   // GBK_TO_UNICODE[12068] := 16#A0D0;
   // GBK_TO_UNICODE[12069] := 16#7298;
   // GBK_TO_UNICODE[12070] := 16#A0D1;
   // GBK_TO_UNICODE[12071] := 16#7299;
   // GBK_TO_UNICODE[12072] := 16#A0D2;
   // GBK_TO_UNICODE[12073] := 16#729A;
   // GBK_TO_UNICODE[12074] := 16#A0D3;
   // GBK_TO_UNICODE[12075] := 16#729B;
   // GBK_TO_UNICODE[12076] := 16#A0D4;
   // GBK_TO_UNICODE[12077] := 16#729C;
   // GBK_TO_UNICODE[12078] := 16#A0D5;
   // GBK_TO_UNICODE[12079] := 16#729D;
   // GBK_TO_UNICODE[12080] := 16#A0D6;
   // GBK_TO_UNICODE[12081] := 16#729E;
   // GBK_TO_UNICODE[12082] := 16#A0D7;
   // GBK_TO_UNICODE[12083] := 16#72A0;
   // GBK_TO_UNICODE[12084] := 16#A0D8;
   // GBK_TO_UNICODE[12085] := 16#72A1;
   // GBK_TO_UNICODE[12086] := 16#A0D9;
   // GBK_TO_UNICODE[12087] := 16#72A2;
   // GBK_TO_UNICODE[12088] := 16#A0DA;
   // GBK_TO_UNICODE[12089] := 16#72A3;
   // GBK_TO_UNICODE[12090] := 16#A0DB;
   // GBK_TO_UNICODE[12091] := 16#72A4;
   // GBK_TO_UNICODE[12092] := 16#A0DC;
   // GBK_TO_UNICODE[12093] := 16#72A5;
   // GBK_TO_UNICODE[12094] := 16#A0DD;
   // GBK_TO_UNICODE[12095] := 16#72A6;
   // GBK_TO_UNICODE[12096] := 16#A0DE;
   // GBK_TO_UNICODE[12097] := 16#72A7;
   // GBK_TO_UNICODE[12098] := 16#A0DF;
   // GBK_TO_UNICODE[12099] := 16#72A8;
   // GBK_TO_UNICODE[12100] := 16#A0E0;
   // GBK_TO_UNICODE[12101] := 16#72A9;
   // GBK_TO_UNICODE[12102] := 16#A0E1;
   // GBK_TO_UNICODE[12103] := 16#72AA;
   // GBK_TO_UNICODE[12104] := 16#A0E2;
   // GBK_TO_UNICODE[12105] := 16#72AB;
   // GBK_TO_UNICODE[12106] := 16#A0E3;
   // GBK_TO_UNICODE[12107] := 16#72AE;
   // GBK_TO_UNICODE[12108] := 16#A0E4;
   // GBK_TO_UNICODE[12109] := 16#72B1;
   // GBK_TO_UNICODE[12110] := 16#A0E5;
   // GBK_TO_UNICODE[12111] := 16#72B2;
   // GBK_TO_UNICODE[12112] := 16#A0E6;
   // GBK_TO_UNICODE[12113] := 16#72B3;
   // GBK_TO_UNICODE[12114] := 16#A0E7;
   // GBK_TO_UNICODE[12115] := 16#72B5;
   // GBK_TO_UNICODE[12116] := 16#A0E8;
   // GBK_TO_UNICODE[12117] := 16#72BA;
   // GBK_TO_UNICODE[12118] := 16#A0E9;
   // GBK_TO_UNICODE[12119] := 16#72BB;
   // GBK_TO_UNICODE[12120] := 16#A0EA;
   // GBK_TO_UNICODE[12121] := 16#72BC;
   // GBK_TO_UNICODE[12122] := 16#A0EB;
   // GBK_TO_UNICODE[12123] := 16#72BD;
   // GBK_TO_UNICODE[12124] := 16#A0EC;
   // GBK_TO_UNICODE[12125] := 16#72BE;
   // GBK_TO_UNICODE[12126] := 16#A0ED;
   // GBK_TO_UNICODE[12127] := 16#72BF;
   // GBK_TO_UNICODE[12128] := 16#A0EE;
   // GBK_TO_UNICODE[12129] := 16#72C0;
   // GBK_TO_UNICODE[12130] := 16#A0EF;
   // GBK_TO_UNICODE[12131] := 16#72C5;
   // GBK_TO_UNICODE[12132] := 16#A0F0;
   // GBK_TO_UNICODE[12133] := 16#72C6;
   // GBK_TO_UNICODE[12134] := 16#A0F1;
   // GBK_TO_UNICODE[12135] := 16#72C7;
   // GBK_TO_UNICODE[12136] := 16#A0F2;
   // GBK_TO_UNICODE[12137] := 16#72C9;
   // GBK_TO_UNICODE[12138] := 16#A0F3;
   // GBK_TO_UNICODE[12139] := 16#72CA;
   // GBK_TO_UNICODE[12140] := 16#A0F4;
   // GBK_TO_UNICODE[12141] := 16#72CB;
   // GBK_TO_UNICODE[12142] := 16#A0F5;
   // GBK_TO_UNICODE[12143] := 16#72CC;
   // GBK_TO_UNICODE[12144] := 16#A0F6;
   // GBK_TO_UNICODE[12145] := 16#72CF;
   // GBK_TO_UNICODE[12146] := 16#A0F7;
   // GBK_TO_UNICODE[12147] := 16#72D1;
   // GBK_TO_UNICODE[12148] := 16#A0F8;
   // GBK_TO_UNICODE[12149] := 16#72D3;
   // GBK_TO_UNICODE[12150] := 16#A0F9;
   // GBK_TO_UNICODE[12151] := 16#72D4;
   // GBK_TO_UNICODE[12152] := 16#A0FA;
   // GBK_TO_UNICODE[12153] := 16#72D5;
   // GBK_TO_UNICODE[12154] := 16#A0FB;
   // GBK_TO_UNICODE[12155] := 16#72D6;
   // GBK_TO_UNICODE[12156] := 16#A0FC;
   // GBK_TO_UNICODE[12157] := 16#72D8;
   // GBK_TO_UNICODE[12158] := 16#A0FD;
   // GBK_TO_UNICODE[12159] := 16#72DA;
   // GBK_TO_UNICODE[12160] := 16#A0FE;
   // GBK_TO_UNICODE[12161] := 16#72DB;
   // GBK_TO_UNICODE[12162] := 16#A1A1;
   // GBK_TO_UNICODE[12163] := 16#3000;
   // GBK_TO_UNICODE[12164] := 16#A1A2;
   // GBK_TO_UNICODE[12165] := 16#3001;
   // GBK_TO_UNICODE[12166] := 16#A1A3;
   // GBK_TO_UNICODE[12167] := 16#3002;
   // GBK_TO_UNICODE[12168] := 16#A1A4;
   // GBK_TO_UNICODE[12169] := 16#00B7;
   // GBK_TO_UNICODE[12170] := 16#A1A5;
   // GBK_TO_UNICODE[12171] := 16#02C9;
   // GBK_TO_UNICODE[12172] := 16#A1A6;
   // GBK_TO_UNICODE[12173] := 16#02C7;
   // GBK_TO_UNICODE[12174] := 16#A1A7;
   // GBK_TO_UNICODE[12175] := 16#00A8;
   // GBK_TO_UNICODE[12176] := 16#A1A8;
   // GBK_TO_UNICODE[12177] := 16#3003;
   // GBK_TO_UNICODE[12178] := 16#A1A9;
   // GBK_TO_UNICODE[12179] := 16#3005;
   // GBK_TO_UNICODE[12180] := 16#A1AA;
   // GBK_TO_UNICODE[12181] := 16#2014;
   // GBK_TO_UNICODE[12182] := 16#A1AB;
   // GBK_TO_UNICODE[12183] := 16#FF5E;
   // GBK_TO_UNICODE[12184] := 16#A1AC;
   // GBK_TO_UNICODE[12185] := 16#2016;
   // GBK_TO_UNICODE[12186] := 16#A1AD;
   // GBK_TO_UNICODE[12187] := 16#2026;
   // GBK_TO_UNICODE[12188] := 16#A1AE;
   // GBK_TO_UNICODE[12189] := 16#2018;
   // GBK_TO_UNICODE[12190] := 16#A1AF;
   // GBK_TO_UNICODE[12191] := 16#2019;
   // GBK_TO_UNICODE[12192] := 16#A1B0;
   // GBK_TO_UNICODE[12193] := 16#201C;
   // GBK_TO_UNICODE[12194] := 16#A1B1;
   // GBK_TO_UNICODE[12195] := 16#201D;
   // GBK_TO_UNICODE[12196] := 16#A1B2;
   // GBK_TO_UNICODE[12197] := 16#3014;
   // GBK_TO_UNICODE[12198] := 16#A1B3;
   // GBK_TO_UNICODE[12199] := 16#3015;
   // GBK_TO_UNICODE[12200] := 16#A1B4;
   // GBK_TO_UNICODE[12201] := 16#3008;
   // GBK_TO_UNICODE[12202] := 16#A1B5;
   // GBK_TO_UNICODE[12203] := 16#3009;
   // GBK_TO_UNICODE[12204] := 16#A1B6;
   // GBK_TO_UNICODE[12205] := 16#300A;
   // GBK_TO_UNICODE[12206] := 16#A1B7;
   // GBK_TO_UNICODE[12207] := 16#300B;
   // GBK_TO_UNICODE[12208] := 16#A1B8;
   // GBK_TO_UNICODE[12209] := 16#300C;
   // GBK_TO_UNICODE[12210] := 16#A1B9;
   // GBK_TO_UNICODE[12211] := 16#300D;
   // GBK_TO_UNICODE[12212] := 16#A1BA;
   // GBK_TO_UNICODE[12213] := 16#300E;
   // GBK_TO_UNICODE[12214] := 16#A1BB;
   // GBK_TO_UNICODE[12215] := 16#300F;
   // GBK_TO_UNICODE[12216] := 16#A1BC;
   // GBK_TO_UNICODE[12217] := 16#3016;
   // GBK_TO_UNICODE[12218] := 16#A1BD;
   // GBK_TO_UNICODE[12219] := 16#3017;
   // GBK_TO_UNICODE[12220] := 16#A1BE;
   // GBK_TO_UNICODE[12221] := 16#3010;
   // GBK_TO_UNICODE[12222] := 16#A1BF;
   // GBK_TO_UNICODE[12223] := 16#3011;
   // GBK_TO_UNICODE[12224] := 16#A1C0;
   // GBK_TO_UNICODE[12225] := 16#00B1;
   // GBK_TO_UNICODE[12226] := 16#A1C1;
   // GBK_TO_UNICODE[12227] := 16#00D7;
   // GBK_TO_UNICODE[12228] := 16#A1C2;
   // GBK_TO_UNICODE[12229] := 16#00F7;
   // GBK_TO_UNICODE[12230] := 16#A1C3;
   // GBK_TO_UNICODE[12231] := 16#2236;
   // GBK_TO_UNICODE[12232] := 16#A1C4;
   // GBK_TO_UNICODE[12233] := 16#2227;
   // GBK_TO_UNICODE[12234] := 16#A1C5;
   // GBK_TO_UNICODE[12235] := 16#2228;
   // GBK_TO_UNICODE[12236] := 16#A1C6;
   // GBK_TO_UNICODE[12237] := 16#2211;
   // GBK_TO_UNICODE[12238] := 16#A1C7;
   // GBK_TO_UNICODE[12239] := 16#220F;
   // GBK_TO_UNICODE[12240] := 16#A1C8;
   // GBK_TO_UNICODE[12241] := 16#222A;
   // GBK_TO_UNICODE[12242] := 16#A1C9;
   // GBK_TO_UNICODE[12243] := 16#2229;
   // GBK_TO_UNICODE[12244] := 16#A1CA;
   // GBK_TO_UNICODE[12245] := 16#2208;
   // GBK_TO_UNICODE[12246] := 16#A1CB;
   // GBK_TO_UNICODE[12247] := 16#2237;
   // GBK_TO_UNICODE[12248] := 16#A1CC;
   // GBK_TO_UNICODE[12249] := 16#221A;
   // GBK_TO_UNICODE[12250] := 16#A1CD;
   // GBK_TO_UNICODE[12251] := 16#22A5;
   // GBK_TO_UNICODE[12252] := 16#A1CE;
   // GBK_TO_UNICODE[12253] := 16#2225;
   // GBK_TO_UNICODE[12254] := 16#A1CF;
   // GBK_TO_UNICODE[12255] := 16#2220;
   // GBK_TO_UNICODE[12256] := 16#A1D0;
   // GBK_TO_UNICODE[12257] := 16#2312;
   // GBK_TO_UNICODE[12258] := 16#A1D1;
   // GBK_TO_UNICODE[12259] := 16#2299;
   // GBK_TO_UNICODE[12260] := 16#A1D2;
   // GBK_TO_UNICODE[12261] := 16#222B;
   // GBK_TO_UNICODE[12262] := 16#A1D3;
   // GBK_TO_UNICODE[12263] := 16#222E;
   // GBK_TO_UNICODE[12264] := 16#A1D4;
   // GBK_TO_UNICODE[12265] := 16#2261;
   // GBK_TO_UNICODE[12266] := 16#A1D5;
   // GBK_TO_UNICODE[12267] := 16#224C;
   // GBK_TO_UNICODE[12268] := 16#A1D6;
   // GBK_TO_UNICODE[12269] := 16#2248;
   // GBK_TO_UNICODE[12270] := 16#A1D7;
   // GBK_TO_UNICODE[12271] := 16#223D;
   // GBK_TO_UNICODE[12272] := 16#A1D8;
   // GBK_TO_UNICODE[12273] := 16#221D;
   // GBK_TO_UNICODE[12274] := 16#A1D9;
   // GBK_TO_UNICODE[12275] := 16#2260;
   // GBK_TO_UNICODE[12276] := 16#A1DA;
   // GBK_TO_UNICODE[12277] := 16#226E;
   // GBK_TO_UNICODE[12278] := 16#A1DB;
   // GBK_TO_UNICODE[12279] := 16#226F;
   // GBK_TO_UNICODE[12280] := 16#A1DC;
   // GBK_TO_UNICODE[12281] := 16#2264;
   // GBK_TO_UNICODE[12282] := 16#A1DD;
   // GBK_TO_UNICODE[12283] := 16#2265;
   // GBK_TO_UNICODE[12284] := 16#A1DE;
   // GBK_TO_UNICODE[12285] := 16#221E;
   // GBK_TO_UNICODE[12286] := 16#A1DF;
   // GBK_TO_UNICODE[12287] := 16#2235;
   // GBK_TO_UNICODE[12288] := 16#A1E0;
   // GBK_TO_UNICODE[12289] := 16#2234;
   // GBK_TO_UNICODE[12290] := 16#A1E1;
   // GBK_TO_UNICODE[12291] := 16#2642;
   // GBK_TO_UNICODE[12292] := 16#A1E2;
   // GBK_TO_UNICODE[12293] := 16#2640;
   // GBK_TO_UNICODE[12294] := 16#A1E3;
   // GBK_TO_UNICODE[12295] := 16#00B0;
   // GBK_TO_UNICODE[12296] := 16#A1E4;
   // GBK_TO_UNICODE[12297] := 16#2032;
   // GBK_TO_UNICODE[12298] := 16#A1E5;
   // GBK_TO_UNICODE[12299] := 16#2033;
   // GBK_TO_UNICODE[12300] := 16#A1E6;
   // GBK_TO_UNICODE[12301] := 16#2103;
   // GBK_TO_UNICODE[12302] := 16#A1E7;
   // GBK_TO_UNICODE[12303] := 16#FF04;
   // GBK_TO_UNICODE[12304] := 16#A1E8;
   // GBK_TO_UNICODE[12305] := 16#00A4;
   // GBK_TO_UNICODE[12306] := 16#A1E9;
   // GBK_TO_UNICODE[12307] := 16#FFE0;
   // GBK_TO_UNICODE[12308] := 16#A1EA;
   // GBK_TO_UNICODE[12309] := 16#FFE1;
   // GBK_TO_UNICODE[12310] := 16#A1EB;
   // GBK_TO_UNICODE[12311] := 16#2030;
   // GBK_TO_UNICODE[12312] := 16#A1EC;
   // GBK_TO_UNICODE[12313] := 16#00A7;
   // GBK_TO_UNICODE[12314] := 16#A1ED;
   // GBK_TO_UNICODE[12315] := 16#2116;
   // GBK_TO_UNICODE[12316] := 16#A1EE;
   // GBK_TO_UNICODE[12317] := 16#2606;
   // GBK_TO_UNICODE[12318] := 16#A1EF;
   // GBK_TO_UNICODE[12319] := 16#2605;
   // GBK_TO_UNICODE[12320] := 16#A1F0;
   // GBK_TO_UNICODE[12321] := 16#25CB;
   // GBK_TO_UNICODE[12322] := 16#A1F1;
   // GBK_TO_UNICODE[12323] := 16#25CF;
   // GBK_TO_UNICODE[12324] := 16#A1F2;
   // GBK_TO_UNICODE[12325] := 16#25CE;
   // GBK_TO_UNICODE[12326] := 16#A1F3;
   // GBK_TO_UNICODE[12327] := 16#25C7;
   // GBK_TO_UNICODE[12328] := 16#A1F4;
   // GBK_TO_UNICODE[12329] := 16#25C6;
   // GBK_TO_UNICODE[12330] := 16#A1F5;
   // GBK_TO_UNICODE[12331] := 16#25A1;
   // GBK_TO_UNICODE[12332] := 16#A1F6;
   // GBK_TO_UNICODE[12333] := 16#25A0;
   // GBK_TO_UNICODE[12334] := 16#A1F7;
   // GBK_TO_UNICODE[12335] := 16#25B3;
   // GBK_TO_UNICODE[12336] := 16#A1F8;
   // GBK_TO_UNICODE[12337] := 16#25B2;
   // GBK_TO_UNICODE[12338] := 16#A1F9;
   // GBK_TO_UNICODE[12339] := 16#203B;
   // GBK_TO_UNICODE[12340] := 16#A1FA;
   // GBK_TO_UNICODE[12341] := 16#2192;
   // GBK_TO_UNICODE[12342] := 16#A1FB;
   // GBK_TO_UNICODE[12343] := 16#2190;
   // GBK_TO_UNICODE[12344] := 16#A1FC;
   // GBK_TO_UNICODE[12345] := 16#2191;
   // GBK_TO_UNICODE[12346] := 16#A1FD;
   // GBK_TO_UNICODE[12347] := 16#2193;
   // GBK_TO_UNICODE[12348] := 16#A1FE;
   // GBK_TO_UNICODE[12349] := 16#3013;
   // GBK_TO_UNICODE[12350] := 16#A2A1;
   // GBK_TO_UNICODE[12351] := 16#2170;
   // GBK_TO_UNICODE[12352] := 16#A2A2;
   // GBK_TO_UNICODE[12353] := 16#2171;
   // GBK_TO_UNICODE[12354] := 16#A2A3;
   // GBK_TO_UNICODE[12355] := 16#2172;
   // GBK_TO_UNICODE[12356] := 16#A2A4;
   // GBK_TO_UNICODE[12357] := 16#2173;
   // GBK_TO_UNICODE[12358] := 16#A2A5;
   // GBK_TO_UNICODE[12359] := 16#2174;
   // GBK_TO_UNICODE[12360] := 16#A2A6;
   // GBK_TO_UNICODE[12361] := 16#2175;
   // GBK_TO_UNICODE[12362] := 16#A2A7;
   // GBK_TO_UNICODE[12363] := 16#2176;
   // GBK_TO_UNICODE[12364] := 16#A2A8;
   // GBK_TO_UNICODE[12365] := 16#2177;
   // GBK_TO_UNICODE[12366] := 16#A2A9;
   // GBK_TO_UNICODE[12367] := 16#2178;
   // GBK_TO_UNICODE[12368] := 16#A2AA;
   // GBK_TO_UNICODE[12369] := 16#2179;
   // GBK_TO_UNICODE[12370] := 16#A2B1;
   // GBK_TO_UNICODE[12371] := 16#2488;
   // GBK_TO_UNICODE[12372] := 16#A2B2;
   // GBK_TO_UNICODE[12373] := 16#2489;
   // GBK_TO_UNICODE[12374] := 16#A2B3;
   // GBK_TO_UNICODE[12375] := 16#248A;
   // GBK_TO_UNICODE[12376] := 16#A2B4;
   // GBK_TO_UNICODE[12377] := 16#248B;
   // GBK_TO_UNICODE[12378] := 16#A2B5;
   // GBK_TO_UNICODE[12379] := 16#248C;
   // GBK_TO_UNICODE[12380] := 16#A2B6;
   // GBK_TO_UNICODE[12381] := 16#248D;
   // GBK_TO_UNICODE[12382] := 16#A2B7;
   // GBK_TO_UNICODE[12383] := 16#248E;
   // GBK_TO_UNICODE[12384] := 16#A2B8;
   // GBK_TO_UNICODE[12385] := 16#248F;
   // GBK_TO_UNICODE[12386] := 16#A2B9;
   // GBK_TO_UNICODE[12387] := 16#2490;
   // GBK_TO_UNICODE[12388] := 16#A2BA;
   // GBK_TO_UNICODE[12389] := 16#2491;
   // GBK_TO_UNICODE[12390] := 16#A2BB;
   // GBK_TO_UNICODE[12391] := 16#2492;
   // GBK_TO_UNICODE[12392] := 16#A2BC;
   // GBK_TO_UNICODE[12393] := 16#2493;
   // GBK_TO_UNICODE[12394] := 16#A2BD;
   // GBK_TO_UNICODE[12395] := 16#2494;
   // GBK_TO_UNICODE[12396] := 16#A2BE;
   // GBK_TO_UNICODE[12397] := 16#2495;
   // GBK_TO_UNICODE[12398] := 16#A2BF;
   // GBK_TO_UNICODE[12399] := 16#2496;
   // GBK_TO_UNICODE[12400] := 16#A2C0;
   // GBK_TO_UNICODE[12401] := 16#2497;
   // GBK_TO_UNICODE[12402] := 16#A2C1;
   // GBK_TO_UNICODE[12403] := 16#2498;
   // GBK_TO_UNICODE[12404] := 16#A2C2;
   // GBK_TO_UNICODE[12405] := 16#2499;
   // GBK_TO_UNICODE[12406] := 16#A2C3;
   // GBK_TO_UNICODE[12407] := 16#249A;
   // GBK_TO_UNICODE[12408] := 16#A2C4;
   // GBK_TO_UNICODE[12409] := 16#249B;
   // GBK_TO_UNICODE[12410] := 16#A2C5;
   // GBK_TO_UNICODE[12411] := 16#2474;
   // GBK_TO_UNICODE[12412] := 16#A2C6;
   // GBK_TO_UNICODE[12413] := 16#2475;
   // GBK_TO_UNICODE[12414] := 16#A2C7;
   // GBK_TO_UNICODE[12415] := 16#2476;
   // GBK_TO_UNICODE[12416] := 16#A2C8;
   // GBK_TO_UNICODE[12417] := 16#2477;
   // GBK_TO_UNICODE[12418] := 16#A2C9;
   // GBK_TO_UNICODE[12419] := 16#2478;
   // GBK_TO_UNICODE[12420] := 16#A2CA;
   // GBK_TO_UNICODE[12421] := 16#2479;
   // GBK_TO_UNICODE[12422] := 16#A2CB;
   // GBK_TO_UNICODE[12423] := 16#247A;
   // GBK_TO_UNICODE[12424] := 16#A2CC;
   // GBK_TO_UNICODE[12425] := 16#247B;
   // GBK_TO_UNICODE[12426] := 16#A2CD;
   // GBK_TO_UNICODE[12427] := 16#247C;
   // GBK_TO_UNICODE[12428] := 16#A2CE;
   // GBK_TO_UNICODE[12429] := 16#247D;
   // GBK_TO_UNICODE[12430] := 16#A2CF;
   // GBK_TO_UNICODE[12431] := 16#247E;
   // GBK_TO_UNICODE[12432] := 16#A2D0;
   // GBK_TO_UNICODE[12433] := 16#247F;
   // GBK_TO_UNICODE[12434] := 16#A2D1;
   // GBK_TO_UNICODE[12435] := 16#2480;
   // GBK_TO_UNICODE[12436] := 16#A2D2;
   // GBK_TO_UNICODE[12437] := 16#2481;
   // GBK_TO_UNICODE[12438] := 16#A2D3;
   // GBK_TO_UNICODE[12439] := 16#2482;
   // GBK_TO_UNICODE[12440] := 16#A2D4;
   // GBK_TO_UNICODE[12441] := 16#2483;
   // GBK_TO_UNICODE[12442] := 16#A2D5;
   // GBK_TO_UNICODE[12443] := 16#2484;
   // GBK_TO_UNICODE[12444] := 16#A2D6;
   // GBK_TO_UNICODE[12445] := 16#2485;
   // GBK_TO_UNICODE[12446] := 16#A2D7;
   // GBK_TO_UNICODE[12447] := 16#2486;
   // GBK_TO_UNICODE[12448] := 16#A2D8;
   // GBK_TO_UNICODE[12449] := 16#2487;
   // GBK_TO_UNICODE[12450] := 16#A2D9;
   // GBK_TO_UNICODE[12451] := 16#2460;
   // GBK_TO_UNICODE[12452] := 16#A2DA;
   // GBK_TO_UNICODE[12453] := 16#2461;
   // GBK_TO_UNICODE[12454] := 16#A2DB;
   // GBK_TO_UNICODE[12455] := 16#2462;
   // GBK_TO_UNICODE[12456] := 16#A2DC;
   // GBK_TO_UNICODE[12457] := 16#2463;
   // GBK_TO_UNICODE[12458] := 16#A2DD;
   // GBK_TO_UNICODE[12459] := 16#2464;
   // GBK_TO_UNICODE[12460] := 16#A2DE;
   // GBK_TO_UNICODE[12461] := 16#2465;
   // GBK_TO_UNICODE[12462] := 16#A2DF;
   // GBK_TO_UNICODE[12463] := 16#2466;
   // GBK_TO_UNICODE[12464] := 16#A2E0;
   // GBK_TO_UNICODE[12465] := 16#2467;
   // GBK_TO_UNICODE[12466] := 16#A2E1;
   // GBK_TO_UNICODE[12467] := 16#2468;
   // GBK_TO_UNICODE[12468] := 16#A2E2;
   // GBK_TO_UNICODE[12469] := 16#2469;
   // GBK_TO_UNICODE[12470] := 16#A2E5;
   // GBK_TO_UNICODE[12471] := 16#3220;
   // GBK_TO_UNICODE[12472] := 16#A2E6;
   // GBK_TO_UNICODE[12473] := 16#3221;
   // GBK_TO_UNICODE[12474] := 16#A2E7;
   // GBK_TO_UNICODE[12475] := 16#3222;
   // GBK_TO_UNICODE[12476] := 16#A2E8;
   // GBK_TO_UNICODE[12477] := 16#3223;
   // GBK_TO_UNICODE[12478] := 16#A2E9;
   // GBK_TO_UNICODE[12479] := 16#3224;
   // GBK_TO_UNICODE[12480] := 16#A2EA;
   // GBK_TO_UNICODE[12481] := 16#3225;
   // GBK_TO_UNICODE[12482] := 16#A2EB;
   // GBK_TO_UNICODE[12483] := 16#3226;
   // GBK_TO_UNICODE[12484] := 16#A2EC;
   // GBK_TO_UNICODE[12485] := 16#3227;
   // GBK_TO_UNICODE[12486] := 16#A2ED;
   // GBK_TO_UNICODE[12487] := 16#3228;
   // GBK_TO_UNICODE[12488] := 16#A2EE;
   // GBK_TO_UNICODE[12489] := 16#3229;
   // GBK_TO_UNICODE[12490] := 16#A2F1;
   // GBK_TO_UNICODE[12491] := 16#2160;
   // GBK_TO_UNICODE[12492] := 16#A2F2;
   // GBK_TO_UNICODE[12493] := 16#2161;
   // GBK_TO_UNICODE[12494] := 16#A2F3;
   // GBK_TO_UNICODE[12495] := 16#2162;
   // GBK_TO_UNICODE[12496] := 16#A2F4;
   // GBK_TO_UNICODE[12497] := 16#2163;
   // GBK_TO_UNICODE[12498] := 16#A2F5;
   // GBK_TO_UNICODE[12499] := 16#2164;
   // GBK_TO_UNICODE[12500] := 16#A2F6;
   // GBK_TO_UNICODE[12501] := 16#2165;
   // GBK_TO_UNICODE[12502] := 16#A2F7;
   // GBK_TO_UNICODE[12503] := 16#2166;
   // GBK_TO_UNICODE[12504] := 16#A2F8;
   // GBK_TO_UNICODE[12505] := 16#2167;
   // GBK_TO_UNICODE[12506] := 16#A2F9;
   // GBK_TO_UNICODE[12507] := 16#2168;
   // GBK_TO_UNICODE[12508] := 16#A2FA;
   // GBK_TO_UNICODE[12509] := 16#2169;
   // GBK_TO_UNICODE[12510] := 16#A2FB;
   // GBK_TO_UNICODE[12511] := 16#216A;
   // GBK_TO_UNICODE[12512] := 16#A2FC;
   // GBK_TO_UNICODE[12513] := 16#216B;
   // GBK_TO_UNICODE[12514] := 16#A3A1;
   // GBK_TO_UNICODE[12515] := 16#FF01;
   // GBK_TO_UNICODE[12516] := 16#A3A2;
   // GBK_TO_UNICODE[12517] := 16#FF02;
   // GBK_TO_UNICODE[12518] := 16#A3A3;
   // GBK_TO_UNICODE[12519] := 16#FF03;
   // GBK_TO_UNICODE[12520] := 16#A3A4;
   // GBK_TO_UNICODE[12521] := 16#FFE5;
   // GBK_TO_UNICODE[12522] := 16#A3A5;
   // GBK_TO_UNICODE[12523] := 16#FF05;
   // GBK_TO_UNICODE[12524] := 16#A3A6;
   // GBK_TO_UNICODE[12525] := 16#FF06;
   // GBK_TO_UNICODE[12526] := 16#A3A7;
   // GBK_TO_UNICODE[12527] := 16#FF07;
   // GBK_TO_UNICODE[12528] := 16#A3A8;
   // GBK_TO_UNICODE[12529] := 16#FF08;
   // GBK_TO_UNICODE[12530] := 16#A3A9;
   // GBK_TO_UNICODE[12531] := 16#FF09;
   // GBK_TO_UNICODE[12532] := 16#A3AA;
   // GBK_TO_UNICODE[12533] := 16#FF0A;
   // GBK_TO_UNICODE[12534] := 16#A3AB;
   // GBK_TO_UNICODE[12535] := 16#FF0B;
   // GBK_TO_UNICODE[12536] := 16#A3AC;
   // GBK_TO_UNICODE[12537] := 16#FF0C;
   // GBK_TO_UNICODE[12538] := 16#A3AD;
   // GBK_TO_UNICODE[12539] := 16#FF0D;
   // GBK_TO_UNICODE[12540] := 16#A3AE;
   // GBK_TO_UNICODE[12541] := 16#FF0E;
   // GBK_TO_UNICODE[12542] := 16#A3AF;
   // GBK_TO_UNICODE[12543] := 16#FF0F;
   // GBK_TO_UNICODE[12544] := 16#A3B0;
   // GBK_TO_UNICODE[12545] := 16#FF10;
   // GBK_TO_UNICODE[12546] := 16#A3B1;
   // GBK_TO_UNICODE[12547] := 16#FF11;
   // GBK_TO_UNICODE[12548] := 16#A3B2;
   // GBK_TO_UNICODE[12549] := 16#FF12;
   // GBK_TO_UNICODE[12550] := 16#A3B3;
   // GBK_TO_UNICODE[12551] := 16#FF13;
   // GBK_TO_UNICODE[12552] := 16#A3B4;
   // GBK_TO_UNICODE[12553] := 16#FF14;
   // GBK_TO_UNICODE[12554] := 16#A3B5;
   // GBK_TO_UNICODE[12555] := 16#FF15;
   // GBK_TO_UNICODE[12556] := 16#A3B6;
   // GBK_TO_UNICODE[12557] := 16#FF16;
   // GBK_TO_UNICODE[12558] := 16#A3B7;
   // GBK_TO_UNICODE[12559] := 16#FF17;
   // GBK_TO_UNICODE[12560] := 16#A3B8;
   // GBK_TO_UNICODE[12561] := 16#FF18;
   // GBK_TO_UNICODE[12562] := 16#A3B9;
   // GBK_TO_UNICODE[12563] := 16#FF19;
   // GBK_TO_UNICODE[12564] := 16#A3BA;
   // GBK_TO_UNICODE[12565] := 16#FF1A;
   // GBK_TO_UNICODE[12566] := 16#A3BB;
   // GBK_TO_UNICODE[12567] := 16#FF1B;
   // GBK_TO_UNICODE[12568] := 16#A3BC;
   // GBK_TO_UNICODE[12569] := 16#FF1C;
   // GBK_TO_UNICODE[12570] := 16#A3BD;
   // GBK_TO_UNICODE[12571] := 16#FF1D;
   // GBK_TO_UNICODE[12572] := 16#A3BE;
   // GBK_TO_UNICODE[12573] := 16#FF1E;
   // GBK_TO_UNICODE[12574] := 16#A3BF;
   // GBK_TO_UNICODE[12575] := 16#FF1F;
   // GBK_TO_UNICODE[12576] := 16#A3C0;
   // GBK_TO_UNICODE[12577] := 16#FF20;
   // GBK_TO_UNICODE[12578] := 16#A3C1;
   // GBK_TO_UNICODE[12579] := 16#FF21;
   // GBK_TO_UNICODE[12580] := 16#A3C2;
   // GBK_TO_UNICODE[12581] := 16#FF22;
   // GBK_TO_UNICODE[12582] := 16#A3C3;
   // GBK_TO_UNICODE[12583] := 16#FF23;
   // GBK_TO_UNICODE[12584] := 16#A3C4;
   // GBK_TO_UNICODE[12585] := 16#FF24;
   // GBK_TO_UNICODE[12586] := 16#A3C5;
   // GBK_TO_UNICODE[12587] := 16#FF25;
   // GBK_TO_UNICODE[12588] := 16#A3C6;
   // GBK_TO_UNICODE[12589] := 16#FF26;
   // GBK_TO_UNICODE[12590] := 16#A3C7;
   // GBK_TO_UNICODE[12591] := 16#FF27;
   // GBK_TO_UNICODE[12592] := 16#A3C8;
   // GBK_TO_UNICODE[12593] := 16#FF28;
   // GBK_TO_UNICODE[12594] := 16#A3C9;
   // GBK_TO_UNICODE[12595] := 16#FF29;
   // GBK_TO_UNICODE[12596] := 16#A3CA;
   // GBK_TO_UNICODE[12597] := 16#FF2A;
   // GBK_TO_UNICODE[12598] := 16#A3CB;
   // GBK_TO_UNICODE[12599] := 16#FF2B;
   // GBK_TO_UNICODE[12600] := 16#A3CC;
   // GBK_TO_UNICODE[12601] := 16#FF2C;
   // GBK_TO_UNICODE[12602] := 16#A3CD;
   // GBK_TO_UNICODE[12603] := 16#FF2D;
   // GBK_TO_UNICODE[12604] := 16#A3CE;
   // GBK_TO_UNICODE[12605] := 16#FF2E;
   // GBK_TO_UNICODE[12606] := 16#A3CF;
   // GBK_TO_UNICODE[12607] := 16#FF2F;
   // GBK_TO_UNICODE[12608] := 16#A3D0;
   // GBK_TO_UNICODE[12609] := 16#FF30;
   // GBK_TO_UNICODE[12610] := 16#A3D1;
   // GBK_TO_UNICODE[12611] := 16#FF31;
   // GBK_TO_UNICODE[12612] := 16#A3D2;
   // GBK_TO_UNICODE[12613] := 16#FF32;
   // GBK_TO_UNICODE[12614] := 16#A3D3;
   // GBK_TO_UNICODE[12615] := 16#FF33;
   // GBK_TO_UNICODE[12616] := 16#A3D4;
   // GBK_TO_UNICODE[12617] := 16#FF34;
   // GBK_TO_UNICODE[12618] := 16#A3D5;
   // GBK_TO_UNICODE[12619] := 16#FF35;
   // GBK_TO_UNICODE[12620] := 16#A3D6;
   // GBK_TO_UNICODE[12621] := 16#FF36;
   // GBK_TO_UNICODE[12622] := 16#A3D7;
   // GBK_TO_UNICODE[12623] := 16#FF37;
   // GBK_TO_UNICODE[12624] := 16#A3D8;
   // GBK_TO_UNICODE[12625] := 16#FF38;
   // GBK_TO_UNICODE[12626] := 16#A3D9;
   // GBK_TO_UNICODE[12627] := 16#FF39;
   // GBK_TO_UNICODE[12628] := 16#A3DA;
   // GBK_TO_UNICODE[12629] := 16#FF3A;
   // GBK_TO_UNICODE[12630] := 16#A3DB;
   // GBK_TO_UNICODE[12631] := 16#FF3B;
   // GBK_TO_UNICODE[12632] := 16#A3DC;
   // GBK_TO_UNICODE[12633] := 16#FF3C;
   // GBK_TO_UNICODE[12634] := 16#A3DD;
   // GBK_TO_UNICODE[12635] := 16#FF3D;
   // GBK_TO_UNICODE[12636] := 16#A3DE;
   // GBK_TO_UNICODE[12637] := 16#FF3E;
   // GBK_TO_UNICODE[12638] := 16#A3DF;
   // GBK_TO_UNICODE[12639] := 16#FF3F;
   // GBK_TO_UNICODE[12640] := 16#A3E0;
   // GBK_TO_UNICODE[12641] := 16#FF40;
   // GBK_TO_UNICODE[12642] := 16#A3E1;
   // GBK_TO_UNICODE[12643] := 16#FF41;
   // GBK_TO_UNICODE[12644] := 16#A3E2;
   // GBK_TO_UNICODE[12645] := 16#FF42;
   // GBK_TO_UNICODE[12646] := 16#A3E3;
   // GBK_TO_UNICODE[12647] := 16#FF43;
   // GBK_TO_UNICODE[12648] := 16#A3E4;
   // GBK_TO_UNICODE[12649] := 16#FF44;
   // GBK_TO_UNICODE[12650] := 16#A3E5;
   // GBK_TO_UNICODE[12651] := 16#FF45;
   // GBK_TO_UNICODE[12652] := 16#A3E6;
   // GBK_TO_UNICODE[12653] := 16#FF46;
   // GBK_TO_UNICODE[12654] := 16#A3E7;
   // GBK_TO_UNICODE[12655] := 16#FF47;
   // GBK_TO_UNICODE[12656] := 16#A3E8;
   // GBK_TO_UNICODE[12657] := 16#FF48;
   // GBK_TO_UNICODE[12658] := 16#A3E9;
   // GBK_TO_UNICODE[12659] := 16#FF49;
   // GBK_TO_UNICODE[12660] := 16#A3EA;
   // GBK_TO_UNICODE[12661] := 16#FF4A;
   // GBK_TO_UNICODE[12662] := 16#A3EB;
   // GBK_TO_UNICODE[12663] := 16#FF4B;
   // GBK_TO_UNICODE[12664] := 16#A3EC;
   // GBK_TO_UNICODE[12665] := 16#FF4C;
   // GBK_TO_UNICODE[12666] := 16#A3ED;
   // GBK_TO_UNICODE[12667] := 16#FF4D;
   // GBK_TO_UNICODE[12668] := 16#A3EE;
   // GBK_TO_UNICODE[12669] := 16#FF4E;
   // GBK_TO_UNICODE[12670] := 16#A3EF;
   // GBK_TO_UNICODE[12671] := 16#FF4F;
   // GBK_TO_UNICODE[12672] := 16#A3F0;
   // GBK_TO_UNICODE[12673] := 16#FF50;
   // GBK_TO_UNICODE[12674] := 16#A3F1;
   // GBK_TO_UNICODE[12675] := 16#FF51;
   // GBK_TO_UNICODE[12676] := 16#A3F2;
   // GBK_TO_UNICODE[12677] := 16#FF52;
   // GBK_TO_UNICODE[12678] := 16#A3F3;
   // GBK_TO_UNICODE[12679] := 16#FF53;
   // GBK_TO_UNICODE[12680] := 16#A3F4;
   // GBK_TO_UNICODE[12681] := 16#FF54;
   // GBK_TO_UNICODE[12682] := 16#A3F5;
   // GBK_TO_UNICODE[12683] := 16#FF55;
   // GBK_TO_UNICODE[12684] := 16#A3F6;
   // GBK_TO_UNICODE[12685] := 16#FF56;
   // GBK_TO_UNICODE[12686] := 16#A3F7;
   // GBK_TO_UNICODE[12687] := 16#FF57;
   // GBK_TO_UNICODE[12688] := 16#A3F8;
   // GBK_TO_UNICODE[12689] := 16#FF58;
   // GBK_TO_UNICODE[12690] := 16#A3F9;
   // GBK_TO_UNICODE[12691] := 16#FF59;
   // GBK_TO_UNICODE[12692] := 16#A3FA;
   // GBK_TO_UNICODE[12693] := 16#FF5A;
   // GBK_TO_UNICODE[12694] := 16#A3FB;
   // GBK_TO_UNICODE[12695] := 16#FF5B;
   // GBK_TO_UNICODE[12696] := 16#A3FC;
   // GBK_TO_UNICODE[12697] := 16#FF5C;
   // GBK_TO_UNICODE[12698] := 16#A3FD;
   // GBK_TO_UNICODE[12699] := 16#FF5D;
   // GBK_TO_UNICODE[12700] := 16#A3FE;
   // GBK_TO_UNICODE[12701] := 16#FFE3;
   // GBK_TO_UNICODE[12702] := 16#A4A1;
   // GBK_TO_UNICODE[12703] := 16#3041;
   // GBK_TO_UNICODE[12704] := 16#A4A2;
   // GBK_TO_UNICODE[12705] := 16#3042;
   // GBK_TO_UNICODE[12706] := 16#A4A3;
   // GBK_TO_UNICODE[12707] := 16#3043;
   // GBK_TO_UNICODE[12708] := 16#A4A4;
   // GBK_TO_UNICODE[12709] := 16#3044;
   // GBK_TO_UNICODE[12710] := 16#A4A5;
   // GBK_TO_UNICODE[12711] := 16#3045;
   // GBK_TO_UNICODE[12712] := 16#A4A6;
   // GBK_TO_UNICODE[12713] := 16#3046;
   // GBK_TO_UNICODE[12714] := 16#A4A7;
   // GBK_TO_UNICODE[12715] := 16#3047;
   // GBK_TO_UNICODE[12716] := 16#A4A8;
   // GBK_TO_UNICODE[12717] := 16#3048;
   // GBK_TO_UNICODE[12718] := 16#A4A9;
   // GBK_TO_UNICODE[12719] := 16#3049;
   // GBK_TO_UNICODE[12720] := 16#A4AA;
   // GBK_TO_UNICODE[12721] := 16#304A;
   // GBK_TO_UNICODE[12722] := 16#A4AB;
   // GBK_TO_UNICODE[12723] := 16#304B;
   // GBK_TO_UNICODE[12724] := 16#A4AC;
   // GBK_TO_UNICODE[12725] := 16#304C;
   // GBK_TO_UNICODE[12726] := 16#A4AD;
   // GBK_TO_UNICODE[12727] := 16#304D;
   // GBK_TO_UNICODE[12728] := 16#A4AE;
   // GBK_TO_UNICODE[12729] := 16#304E;
   // GBK_TO_UNICODE[12730] := 16#A4AF;
   // GBK_TO_UNICODE[12731] := 16#304F;
   // GBK_TO_UNICODE[12732] := 16#A4B0;
   // GBK_TO_UNICODE[12733] := 16#3050;
   // GBK_TO_UNICODE[12734] := 16#A4B1;
   // GBK_TO_UNICODE[12735] := 16#3051;
   // GBK_TO_UNICODE[12736] := 16#A4B2;
   // GBK_TO_UNICODE[12737] := 16#3052;
   // GBK_TO_UNICODE[12738] := 16#A4B3;
   // GBK_TO_UNICODE[12739] := 16#3053;
   // GBK_TO_UNICODE[12740] := 16#A4B4;
   // GBK_TO_UNICODE[12741] := 16#3054;
   // GBK_TO_UNICODE[12742] := 16#A4B5;
   // GBK_TO_UNICODE[12743] := 16#3055;
   // GBK_TO_UNICODE[12744] := 16#A4B6;
   // GBK_TO_UNICODE[12745] := 16#3056;
   // GBK_TO_UNICODE[12746] := 16#A4B7;
   // GBK_TO_UNICODE[12747] := 16#3057;
   // GBK_TO_UNICODE[12748] := 16#A4B8;
   // GBK_TO_UNICODE[12749] := 16#3058;
   // GBK_TO_UNICODE[12750] := 16#A4B9;
   // GBK_TO_UNICODE[12751] := 16#3059;
   // GBK_TO_UNICODE[12752] := 16#A4BA;
   // GBK_TO_UNICODE[12753] := 16#305A;
   // GBK_TO_UNICODE[12754] := 16#A4BB;
   // GBK_TO_UNICODE[12755] := 16#305B;
   // GBK_TO_UNICODE[12756] := 16#A4BC;
   // GBK_TO_UNICODE[12757] := 16#305C;
   // GBK_TO_UNICODE[12758] := 16#A4BD;
   // GBK_TO_UNICODE[12759] := 16#305D;
   // GBK_TO_UNICODE[12760] := 16#A4BE;
   // GBK_TO_UNICODE[12761] := 16#305E;
   // GBK_TO_UNICODE[12762] := 16#A4BF;
   // GBK_TO_UNICODE[12763] := 16#305F;
   // GBK_TO_UNICODE[12764] := 16#A4C0;
   // GBK_TO_UNICODE[12765] := 16#3060;
   // GBK_TO_UNICODE[12766] := 16#A4C1;
   // GBK_TO_UNICODE[12767] := 16#3061;
   // GBK_TO_UNICODE[12768] := 16#A4C2;
   // GBK_TO_UNICODE[12769] := 16#3062;
   // GBK_TO_UNICODE[12770] := 16#A4C3;
   // GBK_TO_UNICODE[12771] := 16#3063;
   // GBK_TO_UNICODE[12772] := 16#A4C4;
   // GBK_TO_UNICODE[12773] := 16#3064;
   // GBK_TO_UNICODE[12774] := 16#A4C5;
   // GBK_TO_UNICODE[12775] := 16#3065;
   // GBK_TO_UNICODE[12776] := 16#A4C6;
   // GBK_TO_UNICODE[12777] := 16#3066;
   // GBK_TO_UNICODE[12778] := 16#A4C7;
   // GBK_TO_UNICODE[12779] := 16#3067;
   // GBK_TO_UNICODE[12780] := 16#A4C8;
   // GBK_TO_UNICODE[12781] := 16#3068;
   // GBK_TO_UNICODE[12782] := 16#A4C9;
   // GBK_TO_UNICODE[12783] := 16#3069;
   // GBK_TO_UNICODE[12784] := 16#A4CA;
   // GBK_TO_UNICODE[12785] := 16#306A;
   // GBK_TO_UNICODE[12786] := 16#A4CB;
   // GBK_TO_UNICODE[12787] := 16#306B;
   // GBK_TO_UNICODE[12788] := 16#A4CC;
   // GBK_TO_UNICODE[12789] := 16#306C;
   // GBK_TO_UNICODE[12790] := 16#A4CD;
   // GBK_TO_UNICODE[12791] := 16#306D;
   // GBK_TO_UNICODE[12792] := 16#A4CE;
   // GBK_TO_UNICODE[12793] := 16#306E;
   // GBK_TO_UNICODE[12794] := 16#A4CF;
   // GBK_TO_UNICODE[12795] := 16#306F;
   // GBK_TO_UNICODE[12796] := 16#A4D0;
   // GBK_TO_UNICODE[12797] := 16#3070;
   // GBK_TO_UNICODE[12798] := 16#A4D1;
   // GBK_TO_UNICODE[12799] := 16#3071;
   // GBK_TO_UNICODE[12800] := 16#A4D2;
   // GBK_TO_UNICODE[12801] := 16#3072;
   // GBK_TO_UNICODE[12802] := 16#A4D3;
   // GBK_TO_UNICODE[12803] := 16#3073;
   // GBK_TO_UNICODE[12804] := 16#A4D4;
   // GBK_TO_UNICODE[12805] := 16#3074;
   // GBK_TO_UNICODE[12806] := 16#A4D5;
   // GBK_TO_UNICODE[12807] := 16#3075;
   // GBK_TO_UNICODE[12808] := 16#A4D6;
   // GBK_TO_UNICODE[12809] := 16#3076;
   // GBK_TO_UNICODE[12810] := 16#A4D7;
   // GBK_TO_UNICODE[12811] := 16#3077;
   // GBK_TO_UNICODE[12812] := 16#A4D8;
   // GBK_TO_UNICODE[12813] := 16#3078;
   // GBK_TO_UNICODE[12814] := 16#A4D9;
   // GBK_TO_UNICODE[12815] := 16#3079;
   // GBK_TO_UNICODE[12816] := 16#A4DA;
   // GBK_TO_UNICODE[12817] := 16#307A;
   // GBK_TO_UNICODE[12818] := 16#A4DB;
   // GBK_TO_UNICODE[12819] := 16#307B;
   // GBK_TO_UNICODE[12820] := 16#A4DC;
   // GBK_TO_UNICODE[12821] := 16#307C;
   // GBK_TO_UNICODE[12822] := 16#A4DD;
   // GBK_TO_UNICODE[12823] := 16#307D;
   // GBK_TO_UNICODE[12824] := 16#A4DE;
   // GBK_TO_UNICODE[12825] := 16#307E;
   // GBK_TO_UNICODE[12826] := 16#A4DF;
   // GBK_TO_UNICODE[12827] := 16#307F;
   // GBK_TO_UNICODE[12828] := 16#A4E0;
   // GBK_TO_UNICODE[12829] := 16#3080;
   // GBK_TO_UNICODE[12830] := 16#A4E1;
   // GBK_TO_UNICODE[12831] := 16#3081;
   // GBK_TO_UNICODE[12832] := 16#A4E2;
   // GBK_TO_UNICODE[12833] := 16#3082;
   // GBK_TO_UNICODE[12834] := 16#A4E3;
   // GBK_TO_UNICODE[12835] := 16#3083;
   // GBK_TO_UNICODE[12836] := 16#A4E4;
   // GBK_TO_UNICODE[12837] := 16#3084;
   // GBK_TO_UNICODE[12838] := 16#A4E5;
   // GBK_TO_UNICODE[12839] := 16#3085;
   // GBK_TO_UNICODE[12840] := 16#A4E6;
   // GBK_TO_UNICODE[12841] := 16#3086;
   // GBK_TO_UNICODE[12842] := 16#A4E7;
   // GBK_TO_UNICODE[12843] := 16#3087;
   // GBK_TO_UNICODE[12844] := 16#A4E8;
   // GBK_TO_UNICODE[12845] := 16#3088;
   // GBK_TO_UNICODE[12846] := 16#A4E9;
   // GBK_TO_UNICODE[12847] := 16#3089;
   // GBK_TO_UNICODE[12848] := 16#A4EA;
   // GBK_TO_UNICODE[12849] := 16#308A;
   // GBK_TO_UNICODE[12850] := 16#A4EB;
   // GBK_TO_UNICODE[12851] := 16#308B;
   // GBK_TO_UNICODE[12852] := 16#A4EC;
   // GBK_TO_UNICODE[12853] := 16#308C;
   // GBK_TO_UNICODE[12854] := 16#A4ED;
   // GBK_TO_UNICODE[12855] := 16#308D;
   // GBK_TO_UNICODE[12856] := 16#A4EE;
   // GBK_TO_UNICODE[12857] := 16#308E;
   // GBK_TO_UNICODE[12858] := 16#A4EF;
   // GBK_TO_UNICODE[12859] := 16#308F;
   // GBK_TO_UNICODE[12860] := 16#A4F0;
   // GBK_TO_UNICODE[12861] := 16#3090;
   // GBK_TO_UNICODE[12862] := 16#A4F1;
   // GBK_TO_UNICODE[12863] := 16#3091;
   // GBK_TO_UNICODE[12864] := 16#A4F2;
   // GBK_TO_UNICODE[12865] := 16#3092;
   // GBK_TO_UNICODE[12866] := 16#A4F3;
   // GBK_TO_UNICODE[12867] := 16#3093;
   // GBK_TO_UNICODE[12868] := 16#A5A1;
   // GBK_TO_UNICODE[12869] := 16#30A1;
   // GBK_TO_UNICODE[12870] := 16#A5A2;
   // GBK_TO_UNICODE[12871] := 16#30A2;
   // GBK_TO_UNICODE[12872] := 16#A5A3;
   // GBK_TO_UNICODE[12873] := 16#30A3;
   // GBK_TO_UNICODE[12874] := 16#A5A4;
   // GBK_TO_UNICODE[12875] := 16#30A4;
   // GBK_TO_UNICODE[12876] := 16#A5A5;
   // GBK_TO_UNICODE[12877] := 16#30A5;
   // GBK_TO_UNICODE[12878] := 16#A5A6;
   // GBK_TO_UNICODE[12879] := 16#30A6;
   // GBK_TO_UNICODE[12880] := 16#A5A7;
   // GBK_TO_UNICODE[12881] := 16#30A7;
   // GBK_TO_UNICODE[12882] := 16#A5A8;
   // GBK_TO_UNICODE[12883] := 16#30A8;
   // GBK_TO_UNICODE[12884] := 16#A5A9;
   // GBK_TO_UNICODE[12885] := 16#30A9;
   // GBK_TO_UNICODE[12886] := 16#A5AA;
   // GBK_TO_UNICODE[12887] := 16#30AA;
   // GBK_TO_UNICODE[12888] := 16#A5AB;
   // GBK_TO_UNICODE[12889] := 16#30AB;
   // GBK_TO_UNICODE[12890] := 16#A5AC;
   // GBK_TO_UNICODE[12891] := 16#30AC;
   // GBK_TO_UNICODE[12892] := 16#A5AD;
   // GBK_TO_UNICODE[12893] := 16#30AD;
   // GBK_TO_UNICODE[12894] := 16#A5AE;
   // GBK_TO_UNICODE[12895] := 16#30AE;
   // GBK_TO_UNICODE[12896] := 16#A5AF;
   // GBK_TO_UNICODE[12897] := 16#30AF;
   // GBK_TO_UNICODE[12898] := 16#A5B0;
   // GBK_TO_UNICODE[12899] := 16#30B0;
   // GBK_TO_UNICODE[12900] := 16#A5B1;
   // GBK_TO_UNICODE[12901] := 16#30B1;
   // GBK_TO_UNICODE[12902] := 16#A5B2;
   // GBK_TO_UNICODE[12903] := 16#30B2;
   // GBK_TO_UNICODE[12904] := 16#A5B3;
   // GBK_TO_UNICODE[12905] := 16#30B3;
   // GBK_TO_UNICODE[12906] := 16#A5B4;
   // GBK_TO_UNICODE[12907] := 16#30B4;
   // GBK_TO_UNICODE[12908] := 16#A5B5;
   // GBK_TO_UNICODE[12909] := 16#30B5;
   // GBK_TO_UNICODE[12910] := 16#A5B6;
   // GBK_TO_UNICODE[12911] := 16#30B6;
   // GBK_TO_UNICODE[12912] := 16#A5B7;
   // GBK_TO_UNICODE[12913] := 16#30B7;
   // GBK_TO_UNICODE[12914] := 16#A5B8;
   // GBK_TO_UNICODE[12915] := 16#30B8;
   // GBK_TO_UNICODE[12916] := 16#A5B9;
   // GBK_TO_UNICODE[12917] := 16#30B9;
   // GBK_TO_UNICODE[12918] := 16#A5BA;
   // GBK_TO_UNICODE[12919] := 16#30BA;
   // GBK_TO_UNICODE[12920] := 16#A5BB;
   // GBK_TO_UNICODE[12921] := 16#30BB;
   // GBK_TO_UNICODE[12922] := 16#A5BC;
   // GBK_TO_UNICODE[12923] := 16#30BC;
   // GBK_TO_UNICODE[12924] := 16#A5BD;
   // GBK_TO_UNICODE[12925] := 16#30BD;
   // GBK_TO_UNICODE[12926] := 16#A5BE;
   // GBK_TO_UNICODE[12927] := 16#30BE;
   // GBK_TO_UNICODE[12928] := 16#A5BF;
   // GBK_TO_UNICODE[12929] := 16#30BF;
   // GBK_TO_UNICODE[12930] := 16#A5C0;
   // GBK_TO_UNICODE[12931] := 16#30C0;
   // GBK_TO_UNICODE[12932] := 16#A5C1;
   // GBK_TO_UNICODE[12933] := 16#30C1;
   // GBK_TO_UNICODE[12934] := 16#A5C2;
   // GBK_TO_UNICODE[12935] := 16#30C2;
   // GBK_TO_UNICODE[12936] := 16#A5C3;
   // GBK_TO_UNICODE[12937] := 16#30C3;
   // GBK_TO_UNICODE[12938] := 16#A5C4;
   // GBK_TO_UNICODE[12939] := 16#30C4;
   // GBK_TO_UNICODE[12940] := 16#A5C5;
   // GBK_TO_UNICODE[12941] := 16#30C5;
   // GBK_TO_UNICODE[12942] := 16#A5C6;
   // GBK_TO_UNICODE[12943] := 16#30C6;
   // GBK_TO_UNICODE[12944] := 16#A5C7;
   // GBK_TO_UNICODE[12945] := 16#30C7;
   // GBK_TO_UNICODE[12946] := 16#A5C8;
   // GBK_TO_UNICODE[12947] := 16#30C8;
   // GBK_TO_UNICODE[12948] := 16#A5C9;
   // GBK_TO_UNICODE[12949] := 16#30C9;
   // GBK_TO_UNICODE[12950] := 16#A5CA;
   // GBK_TO_UNICODE[12951] := 16#30CA;
   // GBK_TO_UNICODE[12952] := 16#A5CB;
   // GBK_TO_UNICODE[12953] := 16#30CB;
   // GBK_TO_UNICODE[12954] := 16#A5CC;
   // GBK_TO_UNICODE[12955] := 16#30CC;
   // GBK_TO_UNICODE[12956] := 16#A5CD;
   // GBK_TO_UNICODE[12957] := 16#30CD;
   // GBK_TO_UNICODE[12958] := 16#A5CE;
   // GBK_TO_UNICODE[12959] := 16#30CE;
   // GBK_TO_UNICODE[12960] := 16#A5CF;
   // GBK_TO_UNICODE[12961] := 16#30CF;
   // GBK_TO_UNICODE[12962] := 16#A5D0;
   // GBK_TO_UNICODE[12963] := 16#30D0;
   // GBK_TO_UNICODE[12964] := 16#A5D1;
   // GBK_TO_UNICODE[12965] := 16#30D1;
   // GBK_TO_UNICODE[12966] := 16#A5D2;
   // GBK_TO_UNICODE[12967] := 16#30D2;
   // GBK_TO_UNICODE[12968] := 16#A5D3;
   // GBK_TO_UNICODE[12969] := 16#30D3;
   // GBK_TO_UNICODE[12970] := 16#A5D4;
   // GBK_TO_UNICODE[12971] := 16#30D4;
   // GBK_TO_UNICODE[12972] := 16#A5D5;
   // GBK_TO_UNICODE[12973] := 16#30D5;
   // GBK_TO_UNICODE[12974] := 16#A5D6;
   // GBK_TO_UNICODE[12975] := 16#30D6;
   // GBK_TO_UNICODE[12976] := 16#A5D7;
   // GBK_TO_UNICODE[12977] := 16#30D7;
   // GBK_TO_UNICODE[12978] := 16#A5D8;
   // GBK_TO_UNICODE[12979] := 16#30D8;
   // GBK_TO_UNICODE[12980] := 16#A5D9;
   // GBK_TO_UNICODE[12981] := 16#30D9;
   // GBK_TO_UNICODE[12982] := 16#A5DA;
   // GBK_TO_UNICODE[12983] := 16#30DA;
   // GBK_TO_UNICODE[12984] := 16#A5DB;
   // GBK_TO_UNICODE[12985] := 16#30DB;
   // GBK_TO_UNICODE[12986] := 16#A5DC;
   // GBK_TO_UNICODE[12987] := 16#30DC;
   // GBK_TO_UNICODE[12988] := 16#A5DD;
   // GBK_TO_UNICODE[12989] := 16#30DD;
   // GBK_TO_UNICODE[12990] := 16#A5DE;
   // GBK_TO_UNICODE[12991] := 16#30DE;
   // GBK_TO_UNICODE[12992] := 16#A5DF;
   // GBK_TO_UNICODE[12993] := 16#30DF;
   // GBK_TO_UNICODE[12994] := 16#A5E0;
   // GBK_TO_UNICODE[12995] := 16#30E0;
   // GBK_TO_UNICODE[12996] := 16#A5E1;
   // GBK_TO_UNICODE[12997] := 16#30E1;
   // GBK_TO_UNICODE[12998] := 16#A5E2;
   // GBK_TO_UNICODE[12999] := 16#30E2;
   // GBK_TO_UNICODE[13000] := 16#A5E3;
   // GBK_TO_UNICODE[13001] := 16#30E3;
   // GBK_TO_UNICODE[13002] := 16#A5E4;
   // GBK_TO_UNICODE[13003] := 16#30E4;
   // GBK_TO_UNICODE[13004] := 16#A5E5;
   // GBK_TO_UNICODE[13005] := 16#30E5;
   // GBK_TO_UNICODE[13006] := 16#A5E6;
   // GBK_TO_UNICODE[13007] := 16#30E6;
   // GBK_TO_UNICODE[13008] := 16#A5E7;
   // GBK_TO_UNICODE[13009] := 16#30E7;
   // GBK_TO_UNICODE[13010] := 16#A5E8;
   // GBK_TO_UNICODE[13011] := 16#30E8;
   // GBK_TO_UNICODE[13012] := 16#A5E9;
   // GBK_TO_UNICODE[13013] := 16#30E9;
   // GBK_TO_UNICODE[13014] := 16#A5EA;
   // GBK_TO_UNICODE[13015] := 16#30EA;
   // GBK_TO_UNICODE[13016] := 16#A5EB;
   // GBK_TO_UNICODE[13017] := 16#30EB;
   // GBK_TO_UNICODE[13018] := 16#A5EC;
   // GBK_TO_UNICODE[13019] := 16#30EC;
   // GBK_TO_UNICODE[13020] := 16#A5ED;
   // GBK_TO_UNICODE[13021] := 16#30ED;
   // GBK_TO_UNICODE[13022] := 16#A5EE;
   // GBK_TO_UNICODE[13023] := 16#30EE;
   // GBK_TO_UNICODE[13024] := 16#A5EF;
   // GBK_TO_UNICODE[13025] := 16#30EF;
   // GBK_TO_UNICODE[13026] := 16#A5F0;
   // GBK_TO_UNICODE[13027] := 16#30F0;
   // GBK_TO_UNICODE[13028] := 16#A5F1;
   // GBK_TO_UNICODE[13029] := 16#30F1;
   // GBK_TO_UNICODE[13030] := 16#A5F2;
   // GBK_TO_UNICODE[13031] := 16#30F2;
   // GBK_TO_UNICODE[13032] := 16#A5F3;
   // GBK_TO_UNICODE[13033] := 16#30F3;
   // GBK_TO_UNICODE[13034] := 16#A5F4;
   // GBK_TO_UNICODE[13035] := 16#30F4;
   // GBK_TO_UNICODE[13036] := 16#A5F5;
   // GBK_TO_UNICODE[13037] := 16#30F5;
   // GBK_TO_UNICODE[13038] := 16#A5F6;
   // GBK_TO_UNICODE[13039] := 16#30F6;
   // GBK_TO_UNICODE[13040] := 16#A6A1;
   // GBK_TO_UNICODE[13041] := 16#0391;
   // GBK_TO_UNICODE[13042] := 16#A6A2;
   // GBK_TO_UNICODE[13043] := 16#0392;
   // GBK_TO_UNICODE[13044] := 16#A6A3;
   // GBK_TO_UNICODE[13045] := 16#0393;
   // GBK_TO_UNICODE[13046] := 16#A6A4;
   // GBK_TO_UNICODE[13047] := 16#0394;
   // GBK_TO_UNICODE[13048] := 16#A6A5;
   // GBK_TO_UNICODE[13049] := 16#0395;
   // GBK_TO_UNICODE[13050] := 16#A6A6;
   // GBK_TO_UNICODE[13051] := 16#0396;
   // GBK_TO_UNICODE[13052] := 16#A6A7;
   // GBK_TO_UNICODE[13053] := 16#0397;
   // GBK_TO_UNICODE[13054] := 16#A6A8;
   // GBK_TO_UNICODE[13055] := 16#0398;
   // GBK_TO_UNICODE[13056] := 16#A6A9;
   // GBK_TO_UNICODE[13057] := 16#0399;
   // GBK_TO_UNICODE[13058] := 16#A6AA;
   // GBK_TO_UNICODE[13059] := 16#039A;
   // GBK_TO_UNICODE[13060] := 16#A6AB;
   // GBK_TO_UNICODE[13061] := 16#039B;
   // GBK_TO_UNICODE[13062] := 16#A6AC;
   // GBK_TO_UNICODE[13063] := 16#039C;
   // GBK_TO_UNICODE[13064] := 16#A6AD;
   // GBK_TO_UNICODE[13065] := 16#039D;
   // GBK_TO_UNICODE[13066] := 16#A6AE;
   // GBK_TO_UNICODE[13067] := 16#039E;
   // GBK_TO_UNICODE[13068] := 16#A6AF;
   // GBK_TO_UNICODE[13069] := 16#039F;
   // GBK_TO_UNICODE[13070] := 16#A6B0;
   // GBK_TO_UNICODE[13071] := 16#03A0;
   // GBK_TO_UNICODE[13072] := 16#A6B1;
   // GBK_TO_UNICODE[13073] := 16#03A1;
   // GBK_TO_UNICODE[13074] := 16#A6B2;
   // GBK_TO_UNICODE[13075] := 16#03A3;
   // GBK_TO_UNICODE[13076] := 16#A6B3;
   // GBK_TO_UNICODE[13077] := 16#03A4;
   // GBK_TO_UNICODE[13078] := 16#A6B4;
   // GBK_TO_UNICODE[13079] := 16#03A5;
   // GBK_TO_UNICODE[13080] := 16#A6B5;
   // GBK_TO_UNICODE[13081] := 16#03A6;
   // GBK_TO_UNICODE[13082] := 16#A6B6;
   // GBK_TO_UNICODE[13083] := 16#03A7;
   // GBK_TO_UNICODE[13084] := 16#A6B7;
   // GBK_TO_UNICODE[13085] := 16#03A8;
   // GBK_TO_UNICODE[13086] := 16#A6B8;
   // GBK_TO_UNICODE[13087] := 16#03A9;
   // GBK_TO_UNICODE[13088] := 16#A6C1;
   // GBK_TO_UNICODE[13089] := 16#03B1;
   // GBK_TO_UNICODE[13090] := 16#A6C2;
   // GBK_TO_UNICODE[13091] := 16#03B2;
   // GBK_TO_UNICODE[13092] := 16#A6C3;
   // GBK_TO_UNICODE[13093] := 16#03B3;
   // GBK_TO_UNICODE[13094] := 16#A6C4;
   // GBK_TO_UNICODE[13095] := 16#03B4;
   // GBK_TO_UNICODE[13096] := 16#A6C5;
   // GBK_TO_UNICODE[13097] := 16#03B5;
   // GBK_TO_UNICODE[13098] := 16#A6C6;
   // GBK_TO_UNICODE[13099] := 16#03B6;
   // GBK_TO_UNICODE[13100] := 16#A6C7;
   // GBK_TO_UNICODE[13101] := 16#03B7;
   // GBK_TO_UNICODE[13102] := 16#A6C8;
   // GBK_TO_UNICODE[13103] := 16#03B8;
   // GBK_TO_UNICODE[13104] := 16#A6C9;
   // GBK_TO_UNICODE[13105] := 16#03B9;
   // GBK_TO_UNICODE[13106] := 16#A6CA;
   // GBK_TO_UNICODE[13107] := 16#03BA;
   // GBK_TO_UNICODE[13108] := 16#A6CB;
   // GBK_TO_UNICODE[13109] := 16#03BB;
   // GBK_TO_UNICODE[13110] := 16#A6CC;
   // GBK_TO_UNICODE[13111] := 16#03BC;
   // GBK_TO_UNICODE[13112] := 16#A6CD;
   // GBK_TO_UNICODE[13113] := 16#03BD;
   // GBK_TO_UNICODE[13114] := 16#A6CE;
   // GBK_TO_UNICODE[13115] := 16#03BE;
   // GBK_TO_UNICODE[13116] := 16#A6CF;
   // GBK_TO_UNICODE[13117] := 16#03BF;
   // GBK_TO_UNICODE[13118] := 16#A6D0;
   // GBK_TO_UNICODE[13119] := 16#03C0;
   // GBK_TO_UNICODE[13120] := 16#A6D1;
   // GBK_TO_UNICODE[13121] := 16#03C1;
   // GBK_TO_UNICODE[13122] := 16#A6D2;
   // GBK_TO_UNICODE[13123] := 16#03C3;
   // GBK_TO_UNICODE[13124] := 16#A6D3;
   // GBK_TO_UNICODE[13125] := 16#03C4;
   // GBK_TO_UNICODE[13126] := 16#A6D4;
   // GBK_TO_UNICODE[13127] := 16#03C5;
   // GBK_TO_UNICODE[13128] := 16#A6D5;
   // GBK_TO_UNICODE[13129] := 16#03C6;
   // GBK_TO_UNICODE[13130] := 16#A6D6;
   // GBK_TO_UNICODE[13131] := 16#03C7;
   // GBK_TO_UNICODE[13132] := 16#A6D7;
   // GBK_TO_UNICODE[13133] := 16#03C8;
   // GBK_TO_UNICODE[13134] := 16#A6D8;
   // GBK_TO_UNICODE[13135] := 16#03C9;
   // GBK_TO_UNICODE[13136] := 16#A6E0;
   // GBK_TO_UNICODE[13137] := 16#FE35;
   // GBK_TO_UNICODE[13138] := 16#A6E1;
   // GBK_TO_UNICODE[13139] := 16#FE36;
   // GBK_TO_UNICODE[13140] := 16#A6E2;
   // GBK_TO_UNICODE[13141] := 16#FE39;
   // GBK_TO_UNICODE[13142] := 16#A6E3;
   // GBK_TO_UNICODE[13143] := 16#FE3A;
   // GBK_TO_UNICODE[13144] := 16#A6E4;
   // GBK_TO_UNICODE[13145] := 16#FE3F;
   // GBK_TO_UNICODE[13146] := 16#A6E5;
   // GBK_TO_UNICODE[13147] := 16#FE40;
   // GBK_TO_UNICODE[13148] := 16#A6E6;
   // GBK_TO_UNICODE[13149] := 16#FE3D;
   // GBK_TO_UNICODE[13150] := 16#A6E7;
   // GBK_TO_UNICODE[13151] := 16#FE3E;
   // GBK_TO_UNICODE[13152] := 16#A6E8;
   // GBK_TO_UNICODE[13153] := 16#FE41;
   // GBK_TO_UNICODE[13154] := 16#A6E9;
   // GBK_TO_UNICODE[13155] := 16#FE42;
   // GBK_TO_UNICODE[13156] := 16#A6EA;
   // GBK_TO_UNICODE[13157] := 16#FE43;
   // GBK_TO_UNICODE[13158] := 16#A6EB;
   // GBK_TO_UNICODE[13159] := 16#FE44;
   // GBK_TO_UNICODE[13160] := 16#A6EE;
   // GBK_TO_UNICODE[13161] := 16#FE3B;
   // GBK_TO_UNICODE[13162] := 16#A6EF;
   // GBK_TO_UNICODE[13163] := 16#FE3C;
   // GBK_TO_UNICODE[13164] := 16#A6F0;
   // GBK_TO_UNICODE[13165] := 16#FE37;
   // GBK_TO_UNICODE[13166] := 16#A6F1;
   // GBK_TO_UNICODE[13167] := 16#FE38;
   // GBK_TO_UNICODE[13168] := 16#A6F2;
   // GBK_TO_UNICODE[13169] := 16#FE31;
   // GBK_TO_UNICODE[13170] := 16#A6F4;
   // GBK_TO_UNICODE[13171] := 16#FE33;
   // GBK_TO_UNICODE[13172] := 16#A6F5;
   // GBK_TO_UNICODE[13173] := 16#FE34;
   // GBK_TO_UNICODE[13174] := 16#A7A1;
   // GBK_TO_UNICODE[13175] := 16#0410;
   // GBK_TO_UNICODE[13176] := 16#A7A2;
   // GBK_TO_UNICODE[13177] := 16#0411;
   // GBK_TO_UNICODE[13178] := 16#A7A3;
   // GBK_TO_UNICODE[13179] := 16#0412;
   // GBK_TO_UNICODE[13180] := 16#A7A4;
   // GBK_TO_UNICODE[13181] := 16#0413;
   // GBK_TO_UNICODE[13182] := 16#A7A5;
   // GBK_TO_UNICODE[13183] := 16#0414;
   // GBK_TO_UNICODE[13184] := 16#A7A6;
   // GBK_TO_UNICODE[13185] := 16#0415;
   // GBK_TO_UNICODE[13186] := 16#A7A7;
   // GBK_TO_UNICODE[13187] := 16#0401;
   // GBK_TO_UNICODE[13188] := 16#A7A8;
   // GBK_TO_UNICODE[13189] := 16#0416;
   // GBK_TO_UNICODE[13190] := 16#A7A9;
   // GBK_TO_UNICODE[13191] := 16#0417;
   // GBK_TO_UNICODE[13192] := 16#A7AA;
   // GBK_TO_UNICODE[13193] := 16#0418;
   // GBK_TO_UNICODE[13194] := 16#A7AB;
   // GBK_TO_UNICODE[13195] := 16#0419;
   // GBK_TO_UNICODE[13196] := 16#A7AC;
   // GBK_TO_UNICODE[13197] := 16#041A;
   // GBK_TO_UNICODE[13198] := 16#A7AD;
   // GBK_TO_UNICODE[13199] := 16#041B;
   // GBK_TO_UNICODE[13200] := 16#A7AE;
   // GBK_TO_UNICODE[13201] := 16#041C;
   // GBK_TO_UNICODE[13202] := 16#A7AF;
   // GBK_TO_UNICODE[13203] := 16#041D;
   // GBK_TO_UNICODE[13204] := 16#A7B0;
   // GBK_TO_UNICODE[13205] := 16#041E;
   // GBK_TO_UNICODE[13206] := 16#A7B1;
   // GBK_TO_UNICODE[13207] := 16#041F;
   // GBK_TO_UNICODE[13208] := 16#A7B2;
   // GBK_TO_UNICODE[13209] := 16#0420;
   // GBK_TO_UNICODE[13210] := 16#A7B3;
   // GBK_TO_UNICODE[13211] := 16#0421;
   // GBK_TO_UNICODE[13212] := 16#A7B4;
   // GBK_TO_UNICODE[13213] := 16#0422;
   // GBK_TO_UNICODE[13214] := 16#A7B5;
   // GBK_TO_UNICODE[13215] := 16#0423;
   // GBK_TO_UNICODE[13216] := 16#A7B6;
   // GBK_TO_UNICODE[13217] := 16#0424;
   // GBK_TO_UNICODE[13218] := 16#A7B7;
   // GBK_TO_UNICODE[13219] := 16#0425;
   // GBK_TO_UNICODE[13220] := 16#A7B8;
   // GBK_TO_UNICODE[13221] := 16#0426;
   // GBK_TO_UNICODE[13222] := 16#A7B9;
   // GBK_TO_UNICODE[13223] := 16#0427;
   // GBK_TO_UNICODE[13224] := 16#A7BA;
   // GBK_TO_UNICODE[13225] := 16#0428;
   // GBK_TO_UNICODE[13226] := 16#A7BB;
   // GBK_TO_UNICODE[13227] := 16#0429;
   // GBK_TO_UNICODE[13228] := 16#A7BC;
   // GBK_TO_UNICODE[13229] := 16#042A;
   // GBK_TO_UNICODE[13230] := 16#A7BD;
   // GBK_TO_UNICODE[13231] := 16#042B;
   // GBK_TO_UNICODE[13232] := 16#A7BE;
   // GBK_TO_UNICODE[13233] := 16#042C;
   // GBK_TO_UNICODE[13234] := 16#A7BF;
   // GBK_TO_UNICODE[13235] := 16#042D;
   // GBK_TO_UNICODE[13236] := 16#A7C0;
   // GBK_TO_UNICODE[13237] := 16#042E;
   // GBK_TO_UNICODE[13238] := 16#A7C1;
   // GBK_TO_UNICODE[13239] := 16#042F;
   // GBK_TO_UNICODE[13240] := 16#A7D1;
   // GBK_TO_UNICODE[13241] := 16#0430;
   // GBK_TO_UNICODE[13242] := 16#A7D2;
   // GBK_TO_UNICODE[13243] := 16#0431;
   // GBK_TO_UNICODE[13244] := 16#A7D3;
   // GBK_TO_UNICODE[13245] := 16#0432;
   // GBK_TO_UNICODE[13246] := 16#A7D4;
   // GBK_TO_UNICODE[13247] := 16#0433;
   // GBK_TO_UNICODE[13248] := 16#A7D5;
   // GBK_TO_UNICODE[13249] := 16#0434;
   // GBK_TO_UNICODE[13250] := 16#A7D6;
   // GBK_TO_UNICODE[13251] := 16#0435;
   // GBK_TO_UNICODE[13252] := 16#A7D7;
   // GBK_TO_UNICODE[13253] := 16#0451;
   // GBK_TO_UNICODE[13254] := 16#A7D8;
   // GBK_TO_UNICODE[13255] := 16#0436;
   // GBK_TO_UNICODE[13256] := 16#A7D9;
   // GBK_TO_UNICODE[13257] := 16#0437;
   // GBK_TO_UNICODE[13258] := 16#A7DA;
   // GBK_TO_UNICODE[13259] := 16#0438;
   // GBK_TO_UNICODE[13260] := 16#A7DB;
   // GBK_TO_UNICODE[13261] := 16#0439;
   // GBK_TO_UNICODE[13262] := 16#A7DC;
   // GBK_TO_UNICODE[13263] := 16#043A;
   // GBK_TO_UNICODE[13264] := 16#A7DD;
   // GBK_TO_UNICODE[13265] := 16#043B;
   // GBK_TO_UNICODE[13266] := 16#A7DE;
   // GBK_TO_UNICODE[13267] := 16#043C;
   // GBK_TO_UNICODE[13268] := 16#A7DF;
   // GBK_TO_UNICODE[13269] := 16#043D;
   // GBK_TO_UNICODE[13270] := 16#A7E0;
   // GBK_TO_UNICODE[13271] := 16#043E;
   // GBK_TO_UNICODE[13272] := 16#A7E1;
   // GBK_TO_UNICODE[13273] := 16#043F;
   // GBK_TO_UNICODE[13274] := 16#A7E2;
   // GBK_TO_UNICODE[13275] := 16#0440;
   // GBK_TO_UNICODE[13276] := 16#A7E3;
   // GBK_TO_UNICODE[13277] := 16#0441;
   // GBK_TO_UNICODE[13278] := 16#A7E4;
   // GBK_TO_UNICODE[13279] := 16#0442;
   // GBK_TO_UNICODE[13280] := 16#A7E5;
   // GBK_TO_UNICODE[13281] := 16#0443;
   // GBK_TO_UNICODE[13282] := 16#A7E6;
   // GBK_TO_UNICODE[13283] := 16#0444;
   // GBK_TO_UNICODE[13284] := 16#A7E7;
   // GBK_TO_UNICODE[13285] := 16#0445;
   // GBK_TO_UNICODE[13286] := 16#A7E8;
   // GBK_TO_UNICODE[13287] := 16#0446;
   // GBK_TO_UNICODE[13288] := 16#A7E9;
   // GBK_TO_UNICODE[13289] := 16#0447;
   // GBK_TO_UNICODE[13290] := 16#A7EA;
   // GBK_TO_UNICODE[13291] := 16#0448;
   // GBK_TO_UNICODE[13292] := 16#A7EB;
   // GBK_TO_UNICODE[13293] := 16#0449;
   // GBK_TO_UNICODE[13294] := 16#A7EC;
   // GBK_TO_UNICODE[13295] := 16#044A;
   // GBK_TO_UNICODE[13296] := 16#A7ED;
   // GBK_TO_UNICODE[13297] := 16#044B;
   // GBK_TO_UNICODE[13298] := 16#A7EE;
   // GBK_TO_UNICODE[13299] := 16#044C;
   // GBK_TO_UNICODE[13300] := 16#A7EF;
   // GBK_TO_UNICODE[13301] := 16#044D;
   // GBK_TO_UNICODE[13302] := 16#A7F0;
   // GBK_TO_UNICODE[13303] := 16#044E;
   // GBK_TO_UNICODE[13304] := 16#A7F1;
   // GBK_TO_UNICODE[13305] := 16#044F;
   // GBK_TO_UNICODE[13306] := 16#A840;
   // GBK_TO_UNICODE[13307] := 16#02CA;
   // GBK_TO_UNICODE[13308] := 16#A841;
   // GBK_TO_UNICODE[13309] := 16#02CB;
   // GBK_TO_UNICODE[13310] := 16#A842;
   // GBK_TO_UNICODE[13311] := 16#02D9;
   // GBK_TO_UNICODE[13312] := 16#A843;
   // GBK_TO_UNICODE[13313] := 16#2013;
   // GBK_TO_UNICODE[13314] := 16#A844;
   // GBK_TO_UNICODE[13315] := 16#2015;
   // GBK_TO_UNICODE[13316] := 16#A845;
   // GBK_TO_UNICODE[13317] := 16#2025;
   // GBK_TO_UNICODE[13318] := 16#A846;
   // GBK_TO_UNICODE[13319] := 16#2035;
   // GBK_TO_UNICODE[13320] := 16#A847;
   // GBK_TO_UNICODE[13321] := 16#2105;
   // GBK_TO_UNICODE[13322] := 16#A848;
   // GBK_TO_UNICODE[13323] := 16#2109;
   // GBK_TO_UNICODE[13324] := 16#A849;
   // GBK_TO_UNICODE[13325] := 16#2196;
   // GBK_TO_UNICODE[13326] := 16#A84A;
   // GBK_TO_UNICODE[13327] := 16#2197;
   // GBK_TO_UNICODE[13328] := 16#A84B;
   // GBK_TO_UNICODE[13329] := 16#2198;
   // GBK_TO_UNICODE[13330] := 16#A84C;
   // GBK_TO_UNICODE[13331] := 16#2199;
   // GBK_TO_UNICODE[13332] := 16#A84D;
   // GBK_TO_UNICODE[13333] := 16#2215;
   // GBK_TO_UNICODE[13334] := 16#A84E;
   // GBK_TO_UNICODE[13335] := 16#221F;
   // GBK_TO_UNICODE[13336] := 16#A84F;
   // GBK_TO_UNICODE[13337] := 16#2223;
   // GBK_TO_UNICODE[13338] := 16#A850;
   // GBK_TO_UNICODE[13339] := 16#2252;
   // GBK_TO_UNICODE[13340] := 16#A851;
   // GBK_TO_UNICODE[13341] := 16#2266;
   // GBK_TO_UNICODE[13342] := 16#A852;
   // GBK_TO_UNICODE[13343] := 16#2267;
   // GBK_TO_UNICODE[13344] := 16#A853;
   // GBK_TO_UNICODE[13345] := 16#22BF;
   // GBK_TO_UNICODE[13346] := 16#A854;
   // GBK_TO_UNICODE[13347] := 16#2550;
   // GBK_TO_UNICODE[13348] := 16#A855;
   // GBK_TO_UNICODE[13349] := 16#2551;
   // GBK_TO_UNICODE[13350] := 16#A856;
   // GBK_TO_UNICODE[13351] := 16#2552;
   // GBK_TO_UNICODE[13352] := 16#A857;
   // GBK_TO_UNICODE[13353] := 16#2553;
   // GBK_TO_UNICODE[13354] := 16#A858;
   // GBK_TO_UNICODE[13355] := 16#2554;
   // GBK_TO_UNICODE[13356] := 16#A859;
   // GBK_TO_UNICODE[13357] := 16#2555;
   // GBK_TO_UNICODE[13358] := 16#A85A;
   // GBK_TO_UNICODE[13359] := 16#2556;
   // GBK_TO_UNICODE[13360] := 16#A85B;
   // GBK_TO_UNICODE[13361] := 16#2557;
   // GBK_TO_UNICODE[13362] := 16#A85C;
   // GBK_TO_UNICODE[13363] := 16#2558;
   // GBK_TO_UNICODE[13364] := 16#A85D;
   // GBK_TO_UNICODE[13365] := 16#2559;
   // GBK_TO_UNICODE[13366] := 16#A85E;
   // GBK_TO_UNICODE[13367] := 16#255A;
   // GBK_TO_UNICODE[13368] := 16#A85F;
   // GBK_TO_UNICODE[13369] := 16#255B;
   // GBK_TO_UNICODE[13370] := 16#A860;
   // GBK_TO_UNICODE[13371] := 16#255C;
   // GBK_TO_UNICODE[13372] := 16#A861;
   // GBK_TO_UNICODE[13373] := 16#255D;
   // GBK_TO_UNICODE[13374] := 16#A862;
   // GBK_TO_UNICODE[13375] := 16#255E;
   // GBK_TO_UNICODE[13376] := 16#A863;
   // GBK_TO_UNICODE[13377] := 16#255F;
   // GBK_TO_UNICODE[13378] := 16#A864;
   // GBK_TO_UNICODE[13379] := 16#2560;
   // GBK_TO_UNICODE[13380] := 16#A865;
   // GBK_TO_UNICODE[13381] := 16#2561;
   // GBK_TO_UNICODE[13382] := 16#A866;
   // GBK_TO_UNICODE[13383] := 16#2562;
   // GBK_TO_UNICODE[13384] := 16#A867;
   // GBK_TO_UNICODE[13385] := 16#2563;
   // GBK_TO_UNICODE[13386] := 16#A868;
   // GBK_TO_UNICODE[13387] := 16#2564;
   // GBK_TO_UNICODE[13388] := 16#A869;
   // GBK_TO_UNICODE[13389] := 16#2565;
   // GBK_TO_UNICODE[13390] := 16#A86A;
   // GBK_TO_UNICODE[13391] := 16#2566;
   // GBK_TO_UNICODE[13392] := 16#A86B;
   // GBK_TO_UNICODE[13393] := 16#2567;
   // GBK_TO_UNICODE[13394] := 16#A86C;
   // GBK_TO_UNICODE[13395] := 16#2568;
   // GBK_TO_UNICODE[13396] := 16#A86D;
   // GBK_TO_UNICODE[13397] := 16#2569;
   // GBK_TO_UNICODE[13398] := 16#A86E;
   // GBK_TO_UNICODE[13399] := 16#256A;
   // GBK_TO_UNICODE[13400] := 16#A86F;
   // GBK_TO_UNICODE[13401] := 16#256B;
   // GBK_TO_UNICODE[13402] := 16#A870;
   // GBK_TO_UNICODE[13403] := 16#256C;
   // GBK_TO_UNICODE[13404] := 16#A871;
   // GBK_TO_UNICODE[13405] := 16#256D;
   // GBK_TO_UNICODE[13406] := 16#A872;
   // GBK_TO_UNICODE[13407] := 16#256E;
   // GBK_TO_UNICODE[13408] := 16#A873;
   // GBK_TO_UNICODE[13409] := 16#256F;
   // GBK_TO_UNICODE[13410] := 16#A874;
   // GBK_TO_UNICODE[13411] := 16#2570;
   // GBK_TO_UNICODE[13412] := 16#A875;
   // GBK_TO_UNICODE[13413] := 16#2571;
   // GBK_TO_UNICODE[13414] := 16#A876;
   // GBK_TO_UNICODE[13415] := 16#2572;
   // GBK_TO_UNICODE[13416] := 16#A877;
   // GBK_TO_UNICODE[13417] := 16#2573;
   // GBK_TO_UNICODE[13418] := 16#A878;
   // GBK_TO_UNICODE[13419] := 16#2581;
   // GBK_TO_UNICODE[13420] := 16#A879;
   // GBK_TO_UNICODE[13421] := 16#2582;
   // GBK_TO_UNICODE[13422] := 16#A87A;
   // GBK_TO_UNICODE[13423] := 16#2583;
   // GBK_TO_UNICODE[13424] := 16#A87B;
   // GBK_TO_UNICODE[13425] := 16#2584;
   // GBK_TO_UNICODE[13426] := 16#A87C;
   // GBK_TO_UNICODE[13427] := 16#2585;
   // GBK_TO_UNICODE[13428] := 16#A87D;
   // GBK_TO_UNICODE[13429] := 16#2586;
   // GBK_TO_UNICODE[13430] := 16#A87E;
   // GBK_TO_UNICODE[13431] := 16#2587;
   // GBK_TO_UNICODE[13432] := 16#A880;
   // GBK_TO_UNICODE[13433] := 16#2588;
   // GBK_TO_UNICODE[13434] := 16#A881;
   // GBK_TO_UNICODE[13435] := 16#2589;
   // GBK_TO_UNICODE[13436] := 16#A882;
   // GBK_TO_UNICODE[13437] := 16#258A;
   // GBK_TO_UNICODE[13438] := 16#A883;
   // GBK_TO_UNICODE[13439] := 16#258B;
   // GBK_TO_UNICODE[13440] := 16#A884;
   // GBK_TO_UNICODE[13441] := 16#258C;
   // GBK_TO_UNICODE[13442] := 16#A885;
   // GBK_TO_UNICODE[13443] := 16#258D;
   // GBK_TO_UNICODE[13444] := 16#A886;
   // GBK_TO_UNICODE[13445] := 16#258E;
   // GBK_TO_UNICODE[13446] := 16#A887;
   // GBK_TO_UNICODE[13447] := 16#258F;
   // GBK_TO_UNICODE[13448] := 16#A888;
   // GBK_TO_UNICODE[13449] := 16#2593;
   // GBK_TO_UNICODE[13450] := 16#A889;
   // GBK_TO_UNICODE[13451] := 16#2594;
   // GBK_TO_UNICODE[13452] := 16#A88A;
   // GBK_TO_UNICODE[13453] := 16#2595;
   // GBK_TO_UNICODE[13454] := 16#A88B;
   // GBK_TO_UNICODE[13455] := 16#25BC;
   // GBK_TO_UNICODE[13456] := 16#A88C;
   // GBK_TO_UNICODE[13457] := 16#25BD;
   // GBK_TO_UNICODE[13458] := 16#A88D;
   // GBK_TO_UNICODE[13459] := 16#25E2;
   // GBK_TO_UNICODE[13460] := 16#A88E;
   // GBK_TO_UNICODE[13461] := 16#25E3;
   // GBK_TO_UNICODE[13462] := 16#A88F;
   // GBK_TO_UNICODE[13463] := 16#25E4;
   // GBK_TO_UNICODE[13464] := 16#A890;
   // GBK_TO_UNICODE[13465] := 16#25E5;
   // GBK_TO_UNICODE[13466] := 16#A891;
   // GBK_TO_UNICODE[13467] := 16#2609;
   // GBK_TO_UNICODE[13468] := 16#A892;
   // GBK_TO_UNICODE[13469] := 16#2295;
   // GBK_TO_UNICODE[13470] := 16#A893;
   // GBK_TO_UNICODE[13471] := 16#3012;
   // GBK_TO_UNICODE[13472] := 16#A894;
   // GBK_TO_UNICODE[13473] := 16#301D;
   // GBK_TO_UNICODE[13474] := 16#A895;
   // GBK_TO_UNICODE[13475] := 16#301E;
   // GBK_TO_UNICODE[13476] := 16#A8A1;
   // GBK_TO_UNICODE[13477] := 16#0101;
   // GBK_TO_UNICODE[13478] := 16#A8A2;
   // GBK_TO_UNICODE[13479] := 16#00E1;
   // GBK_TO_UNICODE[13480] := 16#A8A3;
   // GBK_TO_UNICODE[13481] := 16#01CE;
   // GBK_TO_UNICODE[13482] := 16#A8A4;
   // GBK_TO_UNICODE[13483] := 16#00E0;
   // GBK_TO_UNICODE[13484] := 16#A8A5;
   // GBK_TO_UNICODE[13485] := 16#0113;
   // GBK_TO_UNICODE[13486] := 16#A8A6;
   // GBK_TO_UNICODE[13487] := 16#00E9;
   // GBK_TO_UNICODE[13488] := 16#A8A7;
   // GBK_TO_UNICODE[13489] := 16#011B;
   // GBK_TO_UNICODE[13490] := 16#A8A8;
   // GBK_TO_UNICODE[13491] := 16#00E8;
   // GBK_TO_UNICODE[13492] := 16#A8A9;
   // GBK_TO_UNICODE[13493] := 16#012B;
   // GBK_TO_UNICODE[13494] := 16#A8AA;
   // GBK_TO_UNICODE[13495] := 16#00ED;
   // GBK_TO_UNICODE[13496] := 16#A8AB;
   // GBK_TO_UNICODE[13497] := 16#01D0;
   // GBK_TO_UNICODE[13498] := 16#A8AC;
   // GBK_TO_UNICODE[13499] := 16#00EC;
   // GBK_TO_UNICODE[13500] := 16#A8AD;
   // GBK_TO_UNICODE[13501] := 16#014D;
   // GBK_TO_UNICODE[13502] := 16#A8AE;
   // GBK_TO_UNICODE[13503] := 16#00F3;
   // GBK_TO_UNICODE[13504] := 16#A8AF;
   // GBK_TO_UNICODE[13505] := 16#01D2;
   // GBK_TO_UNICODE[13506] := 16#A8B0;
   // GBK_TO_UNICODE[13507] := 16#00F2;
   // GBK_TO_UNICODE[13508] := 16#A8B1;
   // GBK_TO_UNICODE[13509] := 16#016B;
   // GBK_TO_UNICODE[13510] := 16#A8B2;
   // GBK_TO_UNICODE[13511] := 16#00FA;
   // GBK_TO_UNICODE[13512] := 16#A8B3;
   // GBK_TO_UNICODE[13513] := 16#01D4;
   // GBK_TO_UNICODE[13514] := 16#A8B4;
   // GBK_TO_UNICODE[13515] := 16#00F9;
   // GBK_TO_UNICODE[13516] := 16#A8B5;
   // GBK_TO_UNICODE[13517] := 16#01D6;
   // GBK_TO_UNICODE[13518] := 16#A8B6;
   // GBK_TO_UNICODE[13519] := 16#01D8;
   // GBK_TO_UNICODE[13520] := 16#A8B7;
   // GBK_TO_UNICODE[13521] := 16#01DA;
   // GBK_TO_UNICODE[13522] := 16#A8B8;
   // GBK_TO_UNICODE[13523] := 16#01DC;
   // GBK_TO_UNICODE[13524] := 16#A8B9;
   // GBK_TO_UNICODE[13525] := 16#00FC;
   // GBK_TO_UNICODE[13526] := 16#A8BA;
   // GBK_TO_UNICODE[13527] := 16#00EA;
   // GBK_TO_UNICODE[13528] := 16#A8BB;
   // GBK_TO_UNICODE[13529] := 16#0251;
   // GBK_TO_UNICODE[13530] := 16#A8BD;
   // GBK_TO_UNICODE[13531] := 16#0144;
   // GBK_TO_UNICODE[13532] := 16#A8BE;
   // GBK_TO_UNICODE[13533] := 16#0148;
   // GBK_TO_UNICODE[13534] := 16#A8C0;
   // GBK_TO_UNICODE[13535] := 16#0261;
   // GBK_TO_UNICODE[13536] := 16#A8C5;
   // GBK_TO_UNICODE[13537] := 16#3105;
   // GBK_TO_UNICODE[13538] := 16#A8C6;
   // GBK_TO_UNICODE[13539] := 16#3106;
   // GBK_TO_UNICODE[13540] := 16#A8C7;
   // GBK_TO_UNICODE[13541] := 16#3107;
   // GBK_TO_UNICODE[13542] := 16#A8C8;
   // GBK_TO_UNICODE[13543] := 16#3108;
   // GBK_TO_UNICODE[13544] := 16#A8C9;
   // GBK_TO_UNICODE[13545] := 16#3109;
   // GBK_TO_UNICODE[13546] := 16#A8CA;
   // GBK_TO_UNICODE[13547] := 16#310A;
   // GBK_TO_UNICODE[13548] := 16#A8CB;
   // GBK_TO_UNICODE[13549] := 16#310B;
   // GBK_TO_UNICODE[13550] := 16#A8CC;
   // GBK_TO_UNICODE[13551] := 16#310C;
   // GBK_TO_UNICODE[13552] := 16#A8CD;
   // GBK_TO_UNICODE[13553] := 16#310D;
   // GBK_TO_UNICODE[13554] := 16#A8CE;
   // GBK_TO_UNICODE[13555] := 16#310E;
   // GBK_TO_UNICODE[13556] := 16#A8CF;
   // GBK_TO_UNICODE[13557] := 16#310F;
   // GBK_TO_UNICODE[13558] := 16#A8D0;
   // GBK_TO_UNICODE[13559] := 16#3110;
   // GBK_TO_UNICODE[13560] := 16#A8D1;
   // GBK_TO_UNICODE[13561] := 16#3111;
   // GBK_TO_UNICODE[13562] := 16#A8D2;
   // GBK_TO_UNICODE[13563] := 16#3112;
   // GBK_TO_UNICODE[13564] := 16#A8D3;
   // GBK_TO_UNICODE[13565] := 16#3113;
   // GBK_TO_UNICODE[13566] := 16#A8D4;
   // GBK_TO_UNICODE[13567] := 16#3114;
   // GBK_TO_UNICODE[13568] := 16#A8D5;
   // GBK_TO_UNICODE[13569] := 16#3115;
   // GBK_TO_UNICODE[13570] := 16#A8D6;
   // GBK_TO_UNICODE[13571] := 16#3116;
   // GBK_TO_UNICODE[13572] := 16#A8D7;
   // GBK_TO_UNICODE[13573] := 16#3117;
   // GBK_TO_UNICODE[13574] := 16#A8D8;
   // GBK_TO_UNICODE[13575] := 16#3118;
   // GBK_TO_UNICODE[13576] := 16#A8D9;
   // GBK_TO_UNICODE[13577] := 16#3119;
   // GBK_TO_UNICODE[13578] := 16#A8DA;
   // GBK_TO_UNICODE[13579] := 16#311A;
   // GBK_TO_UNICODE[13580] := 16#A8DB;
   // GBK_TO_UNICODE[13581] := 16#311B;
   // GBK_TO_UNICODE[13582] := 16#A8DC;
   // GBK_TO_UNICODE[13583] := 16#311C;
   // GBK_TO_UNICODE[13584] := 16#A8DD;
   // GBK_TO_UNICODE[13585] := 16#311D;
   // GBK_TO_UNICODE[13586] := 16#A8DE;
   // GBK_TO_UNICODE[13587] := 16#311E;
   // GBK_TO_UNICODE[13588] := 16#A8DF;
   // GBK_TO_UNICODE[13589] := 16#311F;
   // GBK_TO_UNICODE[13590] := 16#A8E0;
   // GBK_TO_UNICODE[13591] := 16#3120;
   // GBK_TO_UNICODE[13592] := 16#A8E1;
   // GBK_TO_UNICODE[13593] := 16#3121;
   // GBK_TO_UNICODE[13594] := 16#A8E2;
   // GBK_TO_UNICODE[13595] := 16#3122;
   // GBK_TO_UNICODE[13596] := 16#A8E3;
   // GBK_TO_UNICODE[13597] := 16#3123;
   // GBK_TO_UNICODE[13598] := 16#A8E4;
   // GBK_TO_UNICODE[13599] := 16#3124;
   // GBK_TO_UNICODE[13600] := 16#A8E5;
   // GBK_TO_UNICODE[13601] := 16#3125;
   // GBK_TO_UNICODE[13602] := 16#A8E6;
   // GBK_TO_UNICODE[13603] := 16#3126;
   // GBK_TO_UNICODE[13604] := 16#A8E7;
   // GBK_TO_UNICODE[13605] := 16#3127;
   // GBK_TO_UNICODE[13606] := 16#A8E8;
   // GBK_TO_UNICODE[13607] := 16#3128;
   // GBK_TO_UNICODE[13608] := 16#A8E9;
   // GBK_TO_UNICODE[13609] := 16#3129;
   // GBK_TO_UNICODE[13610] := 16#A940;
   // GBK_TO_UNICODE[13611] := 16#3021;
   // GBK_TO_UNICODE[13612] := 16#A941;
   // GBK_TO_UNICODE[13613] := 16#3022;
   // GBK_TO_UNICODE[13614] := 16#A942;
   // GBK_TO_UNICODE[13615] := 16#3023;
   // GBK_TO_UNICODE[13616] := 16#A943;
   // GBK_TO_UNICODE[13617] := 16#3024;
   // GBK_TO_UNICODE[13618] := 16#A944;
   // GBK_TO_UNICODE[13619] := 16#3025;
   // GBK_TO_UNICODE[13620] := 16#A945;
   // GBK_TO_UNICODE[13621] := 16#3026;
   // GBK_TO_UNICODE[13622] := 16#A946;
   // GBK_TO_UNICODE[13623] := 16#3027;
   // GBK_TO_UNICODE[13624] := 16#A947;
   // GBK_TO_UNICODE[13625] := 16#3028;
   // GBK_TO_UNICODE[13626] := 16#A948;
   // GBK_TO_UNICODE[13627] := 16#3029;
   // GBK_TO_UNICODE[13628] := 16#A949;
   // GBK_TO_UNICODE[13629] := 16#32A3;
   // GBK_TO_UNICODE[13630] := 16#A94A;
   // GBK_TO_UNICODE[13631] := 16#338E;
   // GBK_TO_UNICODE[13632] := 16#A94B;
   // GBK_TO_UNICODE[13633] := 16#338F;
   // GBK_TO_UNICODE[13634] := 16#A94C;
   // GBK_TO_UNICODE[13635] := 16#339C;
   // GBK_TO_UNICODE[13636] := 16#A94D;
   // GBK_TO_UNICODE[13637] := 16#339D;
   // GBK_TO_UNICODE[13638] := 16#A94E;
   // GBK_TO_UNICODE[13639] := 16#339E;
   // GBK_TO_UNICODE[13640] := 16#A94F;
   // GBK_TO_UNICODE[13641] := 16#33A1;
   // GBK_TO_UNICODE[13642] := 16#A950;
   // GBK_TO_UNICODE[13643] := 16#33C4;
   // GBK_TO_UNICODE[13644] := 16#A951;
   // GBK_TO_UNICODE[13645] := 16#33CE;
   // GBK_TO_UNICODE[13646] := 16#A952;
   // GBK_TO_UNICODE[13647] := 16#33D1;
   // GBK_TO_UNICODE[13648] := 16#A953;
   // GBK_TO_UNICODE[13649] := 16#33D2;
   // GBK_TO_UNICODE[13650] := 16#A954;
   // GBK_TO_UNICODE[13651] := 16#33D5;
   // GBK_TO_UNICODE[13652] := 16#A955;
   // GBK_TO_UNICODE[13653] := 16#FE30;
   // GBK_TO_UNICODE[13654] := 16#A956;
   // GBK_TO_UNICODE[13655] := 16#FFE2;
   // GBK_TO_UNICODE[13656] := 16#A957;
   // GBK_TO_UNICODE[13657] := 16#FFE4;
   // GBK_TO_UNICODE[13658] := 16#A959;
   // GBK_TO_UNICODE[13659] := 16#2121;
   // GBK_TO_UNICODE[13660] := 16#A95A;
   // GBK_TO_UNICODE[13661] := 16#3231;
   // GBK_TO_UNICODE[13662] := 16#A95C;
   // GBK_TO_UNICODE[13663] := 16#2010;
   // GBK_TO_UNICODE[13664] := 16#A960;
   // GBK_TO_UNICODE[13665] := 16#30FC;
   // GBK_TO_UNICODE[13666] := 16#A961;
   // GBK_TO_UNICODE[13667] := 16#309B;
   // GBK_TO_UNICODE[13668] := 16#A962;
   // GBK_TO_UNICODE[13669] := 16#309C;
   // GBK_TO_UNICODE[13670] := 16#A963;
   // GBK_TO_UNICODE[13671] := 16#30FD;
   // GBK_TO_UNICODE[13672] := 16#A964;
   // GBK_TO_UNICODE[13673] := 16#30FE;
   // GBK_TO_UNICODE[13674] := 16#A965;
   // GBK_TO_UNICODE[13675] := 16#3006;
   // GBK_TO_UNICODE[13676] := 16#A966;
   // GBK_TO_UNICODE[13677] := 16#309D;
   // GBK_TO_UNICODE[13678] := 16#A967;
   // GBK_TO_UNICODE[13679] := 16#309E;
   // GBK_TO_UNICODE[13680] := 16#A968;
   // GBK_TO_UNICODE[13681] := 16#FE49;
   // GBK_TO_UNICODE[13682] := 16#A969;
   // GBK_TO_UNICODE[13683] := 16#FE4A;
   // GBK_TO_UNICODE[13684] := 16#A96A;
   // GBK_TO_UNICODE[13685] := 16#FE4B;
   // GBK_TO_UNICODE[13686] := 16#A96B;
   // GBK_TO_UNICODE[13687] := 16#FE4C;
   // GBK_TO_UNICODE[13688] := 16#A96C;
   // GBK_TO_UNICODE[13689] := 16#FE4D;
   // GBK_TO_UNICODE[13690] := 16#A96D;
   // GBK_TO_UNICODE[13691] := 16#FE4E;
   // GBK_TO_UNICODE[13692] := 16#A96E;
   // GBK_TO_UNICODE[13693] := 16#FE4F;
   // GBK_TO_UNICODE[13694] := 16#A96F;
   // GBK_TO_UNICODE[13695] := 16#FE50;
   // GBK_TO_UNICODE[13696] := 16#A970;
   // GBK_TO_UNICODE[13697] := 16#FE51;
   // GBK_TO_UNICODE[13698] := 16#A971;
   // GBK_TO_UNICODE[13699] := 16#FE52;
   // GBK_TO_UNICODE[13700] := 16#A972;
   // GBK_TO_UNICODE[13701] := 16#FE54;
   // GBK_TO_UNICODE[13702] := 16#A973;
   // GBK_TO_UNICODE[13703] := 16#FE55;
   // GBK_TO_UNICODE[13704] := 16#A974;
   // GBK_TO_UNICODE[13705] := 16#FE56;
   // GBK_TO_UNICODE[13706] := 16#A975;
   // GBK_TO_UNICODE[13707] := 16#FE57;
   // GBK_TO_UNICODE[13708] := 16#A976;
   // GBK_TO_UNICODE[13709] := 16#FE59;
   // GBK_TO_UNICODE[13710] := 16#A977;
   // GBK_TO_UNICODE[13711] := 16#FE5A;
   // GBK_TO_UNICODE[13712] := 16#A978;
   // GBK_TO_UNICODE[13713] := 16#FE5B;
   // GBK_TO_UNICODE[13714] := 16#A979;
   // GBK_TO_UNICODE[13715] := 16#FE5C;
   // GBK_TO_UNICODE[13716] := 16#A97A;
   // GBK_TO_UNICODE[13717] := 16#FE5D;
   // GBK_TO_UNICODE[13718] := 16#A97B;
   // GBK_TO_UNICODE[13719] := 16#FE5E;
   // GBK_TO_UNICODE[13720] := 16#A97C;
   // GBK_TO_UNICODE[13721] := 16#FE5F;
   // GBK_TO_UNICODE[13722] := 16#A97D;
   // GBK_TO_UNICODE[13723] := 16#FE60;
   // GBK_TO_UNICODE[13724] := 16#A97E;
   // GBK_TO_UNICODE[13725] := 16#FE61;
   // GBK_TO_UNICODE[13726] := 16#A980;
   // GBK_TO_UNICODE[13727] := 16#FE62;
   // GBK_TO_UNICODE[13728] := 16#A981;
   // GBK_TO_UNICODE[13729] := 16#FE63;
   // GBK_TO_UNICODE[13730] := 16#A982;
   // GBK_TO_UNICODE[13731] := 16#FE64;
   // GBK_TO_UNICODE[13732] := 16#A983;
   // GBK_TO_UNICODE[13733] := 16#FE65;
   // GBK_TO_UNICODE[13734] := 16#A984;
   // GBK_TO_UNICODE[13735] := 16#FE66;
   // GBK_TO_UNICODE[13736] := 16#A985;
   // GBK_TO_UNICODE[13737] := 16#FE68;
   // GBK_TO_UNICODE[13738] := 16#A986;
   // GBK_TO_UNICODE[13739] := 16#FE69;
   // GBK_TO_UNICODE[13740] := 16#A987;
   // GBK_TO_UNICODE[13741] := 16#FE6A;
   // GBK_TO_UNICODE[13742] := 16#A988;
   // GBK_TO_UNICODE[13743] := 16#FE6B;
   // GBK_TO_UNICODE[13744] := 16#A996;
   // GBK_TO_UNICODE[13745] := 16#3007;
   // GBK_TO_UNICODE[13746] := 16#A9A4;
   // GBK_TO_UNICODE[13747] := 16#2500;
   // GBK_TO_UNICODE[13748] := 16#A9A5;
   // GBK_TO_UNICODE[13749] := 16#2501;
   // GBK_TO_UNICODE[13750] := 16#A9A6;
   // GBK_TO_UNICODE[13751] := 16#2502;
   // GBK_TO_UNICODE[13752] := 16#A9A7;
   // GBK_TO_UNICODE[13753] := 16#2503;
   // GBK_TO_UNICODE[13754] := 16#A9A8;
   // GBK_TO_UNICODE[13755] := 16#2504;
   // GBK_TO_UNICODE[13756] := 16#A9A9;
   // GBK_TO_UNICODE[13757] := 16#2505;
   // GBK_TO_UNICODE[13758] := 16#A9AA;
   // GBK_TO_UNICODE[13759] := 16#2506;
   // GBK_TO_UNICODE[13760] := 16#A9AB;
   // GBK_TO_UNICODE[13761] := 16#2507;
   // GBK_TO_UNICODE[13762] := 16#A9AC;
   // GBK_TO_UNICODE[13763] := 16#2508;
   // GBK_TO_UNICODE[13764] := 16#A9AD;
   // GBK_TO_UNICODE[13765] := 16#2509;
   // GBK_TO_UNICODE[13766] := 16#A9AE;
   // GBK_TO_UNICODE[13767] := 16#250A;
   // GBK_TO_UNICODE[13768] := 16#A9AF;
   // GBK_TO_UNICODE[13769] := 16#250B;
   // GBK_TO_UNICODE[13770] := 16#A9B0;
   // GBK_TO_UNICODE[13771] := 16#250C;
   // GBK_TO_UNICODE[13772] := 16#A9B1;
   // GBK_TO_UNICODE[13773] := 16#250D;
   // GBK_TO_UNICODE[13774] := 16#A9B2;
   // GBK_TO_UNICODE[13775] := 16#250E;
   // GBK_TO_UNICODE[13776] := 16#A9B3;
   // GBK_TO_UNICODE[13777] := 16#250F;
   // GBK_TO_UNICODE[13778] := 16#A9B4;
   // GBK_TO_UNICODE[13779] := 16#2510;
   // GBK_TO_UNICODE[13780] := 16#A9B5;
   // GBK_TO_UNICODE[13781] := 16#2511;
   // GBK_TO_UNICODE[13782] := 16#A9B6;
   // GBK_TO_UNICODE[13783] := 16#2512;
   // GBK_TO_UNICODE[13784] := 16#A9B7;
   // GBK_TO_UNICODE[13785] := 16#2513;
   // GBK_TO_UNICODE[13786] := 16#A9B8;
   // GBK_TO_UNICODE[13787] := 16#2514;
   // GBK_TO_UNICODE[13788] := 16#A9B9;
   // GBK_TO_UNICODE[13789] := 16#2515;
   // GBK_TO_UNICODE[13790] := 16#A9BA;
   // GBK_TO_UNICODE[13791] := 16#2516;
   // GBK_TO_UNICODE[13792] := 16#A9BB;
   // GBK_TO_UNICODE[13793] := 16#2517;
   // GBK_TO_UNICODE[13794] := 16#A9BC;
   // GBK_TO_UNICODE[13795] := 16#2518;
   // GBK_TO_UNICODE[13796] := 16#A9BD;
   // GBK_TO_UNICODE[13797] := 16#2519;
   // GBK_TO_UNICODE[13798] := 16#A9BE;
   // GBK_TO_UNICODE[13799] := 16#251A;
   // GBK_TO_UNICODE[13800] := 16#A9BF;
   // GBK_TO_UNICODE[13801] := 16#251B;
   // GBK_TO_UNICODE[13802] := 16#A9C0;
   // GBK_TO_UNICODE[13803] := 16#251C;
   // GBK_TO_UNICODE[13804] := 16#A9C1;
   // GBK_TO_UNICODE[13805] := 16#251D;
   // GBK_TO_UNICODE[13806] := 16#A9C2;
   // GBK_TO_UNICODE[13807] := 16#251E;
   // GBK_TO_UNICODE[13808] := 16#A9C3;
   // GBK_TO_UNICODE[13809] := 16#251F;
   // GBK_TO_UNICODE[13810] := 16#A9C4;
   // GBK_TO_UNICODE[13811] := 16#2520;
   // GBK_TO_UNICODE[13812] := 16#A9C5;
   // GBK_TO_UNICODE[13813] := 16#2521;
   // GBK_TO_UNICODE[13814] := 16#A9C6;
   // GBK_TO_UNICODE[13815] := 16#2522;
   // GBK_TO_UNICODE[13816] := 16#A9C7;
   // GBK_TO_UNICODE[13817] := 16#2523;
   // GBK_TO_UNICODE[13818] := 16#A9C8;
   // GBK_TO_UNICODE[13819] := 16#2524;
   // GBK_TO_UNICODE[13820] := 16#A9C9;
   // GBK_TO_UNICODE[13821] := 16#2525;
   // GBK_TO_UNICODE[13822] := 16#A9CA;
   // GBK_TO_UNICODE[13823] := 16#2526;
   // GBK_TO_UNICODE[13824] := 16#A9CB;
   // GBK_TO_UNICODE[13825] := 16#2527;
   // GBK_TO_UNICODE[13826] := 16#A9CC;
   // GBK_TO_UNICODE[13827] := 16#2528;
   // GBK_TO_UNICODE[13828] := 16#A9CD;
   // GBK_TO_UNICODE[13829] := 16#2529;
   // GBK_TO_UNICODE[13830] := 16#A9CE;
   // GBK_TO_UNICODE[13831] := 16#252A;
   // GBK_TO_UNICODE[13832] := 16#A9CF;
   // GBK_TO_UNICODE[13833] := 16#252B;
   // GBK_TO_UNICODE[13834] := 16#A9D0;
   // GBK_TO_UNICODE[13835] := 16#252C;
   // GBK_TO_UNICODE[13836] := 16#A9D1;
   // GBK_TO_UNICODE[13837] := 16#252D;
   // GBK_TO_UNICODE[13838] := 16#A9D2;
   // GBK_TO_UNICODE[13839] := 16#252E;
   // GBK_TO_UNICODE[13840] := 16#A9D3;
   // GBK_TO_UNICODE[13841] := 16#252F;
   // GBK_TO_UNICODE[13842] := 16#A9D4;
   // GBK_TO_UNICODE[13843] := 16#2530;
   // GBK_TO_UNICODE[13844] := 16#A9D5;
   // GBK_TO_UNICODE[13845] := 16#2531;
   // GBK_TO_UNICODE[13846] := 16#A9D6;
   // GBK_TO_UNICODE[13847] := 16#2532;
   // GBK_TO_UNICODE[13848] := 16#A9D7;
   // GBK_TO_UNICODE[13849] := 16#2533;
   // GBK_TO_UNICODE[13850] := 16#A9D8;
   // GBK_TO_UNICODE[13851] := 16#2534;
   // GBK_TO_UNICODE[13852] := 16#A9D9;
   // GBK_TO_UNICODE[13853] := 16#2535;
   // GBK_TO_UNICODE[13854] := 16#A9DA;
   // GBK_TO_UNICODE[13855] := 16#2536;
   // GBK_TO_UNICODE[13856] := 16#A9DB;
   // GBK_TO_UNICODE[13857] := 16#2537;
   // GBK_TO_UNICODE[13858] := 16#A9DC;
   // GBK_TO_UNICODE[13859] := 16#2538;
   // GBK_TO_UNICODE[13860] := 16#A9DD;
   // GBK_TO_UNICODE[13861] := 16#2539;
   // GBK_TO_UNICODE[13862] := 16#A9DE;
   // GBK_TO_UNICODE[13863] := 16#253A;
   // GBK_TO_UNICODE[13864] := 16#A9DF;
   // GBK_TO_UNICODE[13865] := 16#253B;
   // GBK_TO_UNICODE[13866] := 16#A9E0;
   // GBK_TO_UNICODE[13867] := 16#253C;
   // GBK_TO_UNICODE[13868] := 16#A9E1;
   // GBK_TO_UNICODE[13869] := 16#253D;
   // GBK_TO_UNICODE[13870] := 16#A9E2;
   // GBK_TO_UNICODE[13871] := 16#253E;
   // GBK_TO_UNICODE[13872] := 16#A9E3;
   // GBK_TO_UNICODE[13873] := 16#253F;
   // GBK_TO_UNICODE[13874] := 16#A9E4;
   // GBK_TO_UNICODE[13875] := 16#2540;
   // GBK_TO_UNICODE[13876] := 16#A9E5;
   // GBK_TO_UNICODE[13877] := 16#2541;
   // GBK_TO_UNICODE[13878] := 16#A9E6;
   // GBK_TO_UNICODE[13879] := 16#2542;
   // GBK_TO_UNICODE[13880] := 16#A9E7;
   // GBK_TO_UNICODE[13881] := 16#2543;
   // GBK_TO_UNICODE[13882] := 16#A9E8;
   // GBK_TO_UNICODE[13883] := 16#2544;
   // GBK_TO_UNICODE[13884] := 16#A9E9;
   // GBK_TO_UNICODE[13885] := 16#2545;
   // GBK_TO_UNICODE[13886] := 16#A9EA;
   // GBK_TO_UNICODE[13887] := 16#2546;
   // GBK_TO_UNICODE[13888] := 16#A9EB;
   // GBK_TO_UNICODE[13889] := 16#2547;
   // GBK_TO_UNICODE[13890] := 16#A9EC;
   // GBK_TO_UNICODE[13891] := 16#2548;
   // GBK_TO_UNICODE[13892] := 16#A9ED;
   // GBK_TO_UNICODE[13893] := 16#2549;
   // GBK_TO_UNICODE[13894] := 16#A9EE;
   // GBK_TO_UNICODE[13895] := 16#254A;
   // GBK_TO_UNICODE[13896] := 16#A9EF;
   // GBK_TO_UNICODE[13897] := 16#254B;
   // GBK_TO_UNICODE[13898] := 16#AA40;
   // GBK_TO_UNICODE[13899] := 16#72DC;
   // GBK_TO_UNICODE[13900] := 16#AA41;
   // GBK_TO_UNICODE[13901] := 16#72DD;
   // GBK_TO_UNICODE[13902] := 16#AA42;
   // GBK_TO_UNICODE[13903] := 16#72DF;
   // GBK_TO_UNICODE[13904] := 16#AA43;
   // GBK_TO_UNICODE[13905] := 16#72E2;
   // GBK_TO_UNICODE[13906] := 16#AA44;
   // GBK_TO_UNICODE[13907] := 16#72E3;
   // GBK_TO_UNICODE[13908] := 16#AA45;
   // GBK_TO_UNICODE[13909] := 16#72E4;
   // GBK_TO_UNICODE[13910] := 16#AA46;
   // GBK_TO_UNICODE[13911] := 16#72E5;
   // GBK_TO_UNICODE[13912] := 16#AA47;
   // GBK_TO_UNICODE[13913] := 16#72E6;
   // GBK_TO_UNICODE[13914] := 16#AA48;
   // GBK_TO_UNICODE[13915] := 16#72E7;
   // GBK_TO_UNICODE[13916] := 16#AA49;
   // GBK_TO_UNICODE[13917] := 16#72EA;
   // GBK_TO_UNICODE[13918] := 16#AA4A;
   // GBK_TO_UNICODE[13919] := 16#72EB;
   // GBK_TO_UNICODE[13920] := 16#AA4B;
   // GBK_TO_UNICODE[13921] := 16#72F5;
   // GBK_TO_UNICODE[13922] := 16#AA4C;
   // GBK_TO_UNICODE[13923] := 16#72F6;
   // GBK_TO_UNICODE[13924] := 16#AA4D;
   // GBK_TO_UNICODE[13925] := 16#72F9;
   // GBK_TO_UNICODE[13926] := 16#AA4E;
   // GBK_TO_UNICODE[13927] := 16#72FD;
   // GBK_TO_UNICODE[13928] := 16#AA4F;
   // GBK_TO_UNICODE[13929] := 16#72FE;
   // GBK_TO_UNICODE[13930] := 16#AA50;
   // GBK_TO_UNICODE[13931] := 16#72FF;
   // GBK_TO_UNICODE[13932] := 16#AA51;
   // GBK_TO_UNICODE[13933] := 16#7300;
   // GBK_TO_UNICODE[13934] := 16#AA52;
   // GBK_TO_UNICODE[13935] := 16#7302;
   // GBK_TO_UNICODE[13936] := 16#AA53;
   // GBK_TO_UNICODE[13937] := 16#7304;
   // GBK_TO_UNICODE[13938] := 16#AA54;
   // GBK_TO_UNICODE[13939] := 16#7305;
   // GBK_TO_UNICODE[13940] := 16#AA55;
   // GBK_TO_UNICODE[13941] := 16#7306;
   // GBK_TO_UNICODE[13942] := 16#AA56;
   // GBK_TO_UNICODE[13943] := 16#7307;
   // GBK_TO_UNICODE[13944] := 16#AA57;
   // GBK_TO_UNICODE[13945] := 16#7308;
   // GBK_TO_UNICODE[13946] := 16#AA58;
   // GBK_TO_UNICODE[13947] := 16#7309;
   // GBK_TO_UNICODE[13948] := 16#AA59;
   // GBK_TO_UNICODE[13949] := 16#730B;
   // GBK_TO_UNICODE[13950] := 16#AA5A;
   // GBK_TO_UNICODE[13951] := 16#730C;
   // GBK_TO_UNICODE[13952] := 16#AA5B;
   // GBK_TO_UNICODE[13953] := 16#730D;
   // GBK_TO_UNICODE[13954] := 16#AA5C;
   // GBK_TO_UNICODE[13955] := 16#730F;
   // GBK_TO_UNICODE[13956] := 16#AA5D;
   // GBK_TO_UNICODE[13957] := 16#7310;
   // GBK_TO_UNICODE[13958] := 16#AA5E;
   // GBK_TO_UNICODE[13959] := 16#7311;
   // GBK_TO_UNICODE[13960] := 16#AA5F;
   // GBK_TO_UNICODE[13961] := 16#7312;
   // GBK_TO_UNICODE[13962] := 16#AA60;
   // GBK_TO_UNICODE[13963] := 16#7314;
   // GBK_TO_UNICODE[13964] := 16#AA61;
   // GBK_TO_UNICODE[13965] := 16#7318;
   // GBK_TO_UNICODE[13966] := 16#AA62;
   // GBK_TO_UNICODE[13967] := 16#7319;
   // GBK_TO_UNICODE[13968] := 16#AA63;
   // GBK_TO_UNICODE[13969] := 16#731A;
   // GBK_TO_UNICODE[13970] := 16#AA64;
   // GBK_TO_UNICODE[13971] := 16#731F;
   // GBK_TO_UNICODE[13972] := 16#AA65;
   // GBK_TO_UNICODE[13973] := 16#7320;
   // GBK_TO_UNICODE[13974] := 16#AA66;
   // GBK_TO_UNICODE[13975] := 16#7323;
   // GBK_TO_UNICODE[13976] := 16#AA67;
   // GBK_TO_UNICODE[13977] := 16#7324;
   // GBK_TO_UNICODE[13978] := 16#AA68;
   // GBK_TO_UNICODE[13979] := 16#7326;
   // GBK_TO_UNICODE[13980] := 16#AA69;
   // GBK_TO_UNICODE[13981] := 16#7327;
   // GBK_TO_UNICODE[13982] := 16#AA6A;
   // GBK_TO_UNICODE[13983] := 16#7328;
   // GBK_TO_UNICODE[13984] := 16#AA6B;
   // GBK_TO_UNICODE[13985] := 16#732D;
   // GBK_TO_UNICODE[13986] := 16#AA6C;
   // GBK_TO_UNICODE[13987] := 16#732F;
   // GBK_TO_UNICODE[13988] := 16#AA6D;
   // GBK_TO_UNICODE[13989] := 16#7330;
   // GBK_TO_UNICODE[13990] := 16#AA6E;
   // GBK_TO_UNICODE[13991] := 16#7332;
   // GBK_TO_UNICODE[13992] := 16#AA6F;
   // GBK_TO_UNICODE[13993] := 16#7333;
   // GBK_TO_UNICODE[13994] := 16#AA70;
   // GBK_TO_UNICODE[13995] := 16#7335;
   // GBK_TO_UNICODE[13996] := 16#AA71;
   // GBK_TO_UNICODE[13997] := 16#7336;
   // GBK_TO_UNICODE[13998] := 16#AA72;
   // GBK_TO_UNICODE[13999] := 16#733A;
   // GBK_TO_UNICODE[14000] := 16#AA73;
   // GBK_TO_UNICODE[14001] := 16#733B;
   // GBK_TO_UNICODE[14002] := 16#AA74;
   // GBK_TO_UNICODE[14003] := 16#733C;
   // GBK_TO_UNICODE[14004] := 16#AA75;
   // GBK_TO_UNICODE[14005] := 16#733D;
   // GBK_TO_UNICODE[14006] := 16#AA76;
   // GBK_TO_UNICODE[14007] := 16#7340;
   // GBK_TO_UNICODE[14008] := 16#AA77;
   // GBK_TO_UNICODE[14009] := 16#7341;
   // GBK_TO_UNICODE[14010] := 16#AA78;
   // GBK_TO_UNICODE[14011] := 16#7342;
   // GBK_TO_UNICODE[14012] := 16#AA79;
   // GBK_TO_UNICODE[14013] := 16#7343;
   // GBK_TO_UNICODE[14014] := 16#AA7A;
   // GBK_TO_UNICODE[14015] := 16#7344;
   // GBK_TO_UNICODE[14016] := 16#AA7B;
   // GBK_TO_UNICODE[14017] := 16#7345;
   // GBK_TO_UNICODE[14018] := 16#AA7C;
   // GBK_TO_UNICODE[14019] := 16#7346;
   // GBK_TO_UNICODE[14020] := 16#AA7D;
   // GBK_TO_UNICODE[14021] := 16#7347;
   // GBK_TO_UNICODE[14022] := 16#AA7E;
   // GBK_TO_UNICODE[14023] := 16#7348;
   // GBK_TO_UNICODE[14024] := 16#AA80;
   // GBK_TO_UNICODE[14025] := 16#7349;
   // GBK_TO_UNICODE[14026] := 16#AA81;
   // GBK_TO_UNICODE[14027] := 16#734A;
   // GBK_TO_UNICODE[14028] := 16#AA82;
   // GBK_TO_UNICODE[14029] := 16#734B;
   // GBK_TO_UNICODE[14030] := 16#AA83;
   // GBK_TO_UNICODE[14031] := 16#734C;
   // GBK_TO_UNICODE[14032] := 16#AA84;
   // GBK_TO_UNICODE[14033] := 16#734E;
   // GBK_TO_UNICODE[14034] := 16#AA85;
   // GBK_TO_UNICODE[14035] := 16#734F;
   // GBK_TO_UNICODE[14036] := 16#AA86;
   // GBK_TO_UNICODE[14037] := 16#7351;
   // GBK_TO_UNICODE[14038] := 16#AA87;
   // GBK_TO_UNICODE[14039] := 16#7353;
   // GBK_TO_UNICODE[14040] := 16#AA88;
   // GBK_TO_UNICODE[14041] := 16#7354;
   // GBK_TO_UNICODE[14042] := 16#AA89;
   // GBK_TO_UNICODE[14043] := 16#7355;
   // GBK_TO_UNICODE[14044] := 16#AA8A;
   // GBK_TO_UNICODE[14045] := 16#7356;
   // GBK_TO_UNICODE[14046] := 16#AA8B;
   // GBK_TO_UNICODE[14047] := 16#7358;
   // GBK_TO_UNICODE[14048] := 16#AA8C;
   // GBK_TO_UNICODE[14049] := 16#7359;
   // GBK_TO_UNICODE[14050] := 16#AA8D;
   // GBK_TO_UNICODE[14051] := 16#735A;
   // GBK_TO_UNICODE[14052] := 16#AA8E;
   // GBK_TO_UNICODE[14053] := 16#735B;
   // GBK_TO_UNICODE[14054] := 16#AA8F;
   // GBK_TO_UNICODE[14055] := 16#735C;
   // GBK_TO_UNICODE[14056] := 16#AA90;
   // GBK_TO_UNICODE[14057] := 16#735D;
   // GBK_TO_UNICODE[14058] := 16#AA91;
   // GBK_TO_UNICODE[14059] := 16#735E;
   // GBK_TO_UNICODE[14060] := 16#AA92;
   // GBK_TO_UNICODE[14061] := 16#735F;
   // GBK_TO_UNICODE[14062] := 16#AA93;
   // GBK_TO_UNICODE[14063] := 16#7361;
   // GBK_TO_UNICODE[14064] := 16#AA94;
   // GBK_TO_UNICODE[14065] := 16#7362;
   // GBK_TO_UNICODE[14066] := 16#AA95;
   // GBK_TO_UNICODE[14067] := 16#7363;
   // GBK_TO_UNICODE[14068] := 16#AA96;
   // GBK_TO_UNICODE[14069] := 16#7364;
   // GBK_TO_UNICODE[14070] := 16#AA97;
   // GBK_TO_UNICODE[14071] := 16#7365;
   // GBK_TO_UNICODE[14072] := 16#AA98;
   // GBK_TO_UNICODE[14073] := 16#7366;
   // GBK_TO_UNICODE[14074] := 16#AA99;
   // GBK_TO_UNICODE[14075] := 16#7367;
   // GBK_TO_UNICODE[14076] := 16#AA9A;
   // GBK_TO_UNICODE[14077] := 16#7368;
   // GBK_TO_UNICODE[14078] := 16#AA9B;
   // GBK_TO_UNICODE[14079] := 16#7369;
   // GBK_TO_UNICODE[14080] := 16#AA9C;
   // GBK_TO_UNICODE[14081] := 16#736A;
   // GBK_TO_UNICODE[14082] := 16#AA9D;
   // GBK_TO_UNICODE[14083] := 16#736B;
   // GBK_TO_UNICODE[14084] := 16#AA9E;
   // GBK_TO_UNICODE[14085] := 16#736E;
   // GBK_TO_UNICODE[14086] := 16#AA9F;
   // GBK_TO_UNICODE[14087] := 16#7370;
   // GBK_TO_UNICODE[14088] := 16#AAA0;
   // GBK_TO_UNICODE[14089] := 16#7371;
   // GBK_TO_UNICODE[14090] := 16#AB40;
   // GBK_TO_UNICODE[14091] := 16#7372;
   // GBK_TO_UNICODE[14092] := 16#AB41;
   // GBK_TO_UNICODE[14093] := 16#7373;
   // GBK_TO_UNICODE[14094] := 16#AB42;
   // GBK_TO_UNICODE[14095] := 16#7374;
   // GBK_TO_UNICODE[14096] := 16#AB43;
   // GBK_TO_UNICODE[14097] := 16#7375;
   // GBK_TO_UNICODE[14098] := 16#AB44;
   // GBK_TO_UNICODE[14099] := 16#7376;
   // GBK_TO_UNICODE[14100] := 16#AB45;
   // GBK_TO_UNICODE[14101] := 16#7377;
   // GBK_TO_UNICODE[14102] := 16#AB46;
   // GBK_TO_UNICODE[14103] := 16#7378;
   // GBK_TO_UNICODE[14104] := 16#AB47;
   // GBK_TO_UNICODE[14105] := 16#7379;
   // GBK_TO_UNICODE[14106] := 16#AB48;
   // GBK_TO_UNICODE[14107] := 16#737A;
   // GBK_TO_UNICODE[14108] := 16#AB49;
   // GBK_TO_UNICODE[14109] := 16#737B;
   // GBK_TO_UNICODE[14110] := 16#AB4A;
   // GBK_TO_UNICODE[14111] := 16#737C;
   // GBK_TO_UNICODE[14112] := 16#AB4B;
   // GBK_TO_UNICODE[14113] := 16#737D;
   // GBK_TO_UNICODE[14114] := 16#AB4C;
   // GBK_TO_UNICODE[14115] := 16#737F;
   // GBK_TO_UNICODE[14116] := 16#AB4D;
   // GBK_TO_UNICODE[14117] := 16#7380;
   // GBK_TO_UNICODE[14118] := 16#AB4E;
   // GBK_TO_UNICODE[14119] := 16#7381;
   // GBK_TO_UNICODE[14120] := 16#AB4F;
   // GBK_TO_UNICODE[14121] := 16#7382;
   // GBK_TO_UNICODE[14122] := 16#AB50;
   // GBK_TO_UNICODE[14123] := 16#7383;
   // GBK_TO_UNICODE[14124] := 16#AB51;
   // GBK_TO_UNICODE[14125] := 16#7385;
   // GBK_TO_UNICODE[14126] := 16#AB52;
   // GBK_TO_UNICODE[14127] := 16#7386;
   // GBK_TO_UNICODE[14128] := 16#AB53;
   // GBK_TO_UNICODE[14129] := 16#7388;
   // GBK_TO_UNICODE[14130] := 16#AB54;
   // GBK_TO_UNICODE[14131] := 16#738A;
   // GBK_TO_UNICODE[14132] := 16#AB55;
   // GBK_TO_UNICODE[14133] := 16#738C;
   // GBK_TO_UNICODE[14134] := 16#AB56;
   // GBK_TO_UNICODE[14135] := 16#738D;
   // GBK_TO_UNICODE[14136] := 16#AB57;
   // GBK_TO_UNICODE[14137] := 16#738F;
   // GBK_TO_UNICODE[14138] := 16#AB58;
   // GBK_TO_UNICODE[14139] := 16#7390;
   // GBK_TO_UNICODE[14140] := 16#AB59;
   // GBK_TO_UNICODE[14141] := 16#7392;
   // GBK_TO_UNICODE[14142] := 16#AB5A;
   // GBK_TO_UNICODE[14143] := 16#7393;
   // GBK_TO_UNICODE[14144] := 16#AB5B;
   // GBK_TO_UNICODE[14145] := 16#7394;
   // GBK_TO_UNICODE[14146] := 16#AB5C;
   // GBK_TO_UNICODE[14147] := 16#7395;
   // GBK_TO_UNICODE[14148] := 16#AB5D;
   // GBK_TO_UNICODE[14149] := 16#7397;
   // GBK_TO_UNICODE[14150] := 16#AB5E;
   // GBK_TO_UNICODE[14151] := 16#7398;
   // GBK_TO_UNICODE[14152] := 16#AB5F;
   // GBK_TO_UNICODE[14153] := 16#7399;
   // GBK_TO_UNICODE[14154] := 16#AB60;
   // GBK_TO_UNICODE[14155] := 16#739A;
   // GBK_TO_UNICODE[14156] := 16#AB61;
   // GBK_TO_UNICODE[14157] := 16#739C;
   // GBK_TO_UNICODE[14158] := 16#AB62;
   // GBK_TO_UNICODE[14159] := 16#739D;
   // GBK_TO_UNICODE[14160] := 16#AB63;
   // GBK_TO_UNICODE[14161] := 16#739E;
   // GBK_TO_UNICODE[14162] := 16#AB64;
   // GBK_TO_UNICODE[14163] := 16#73A0;
   // GBK_TO_UNICODE[14164] := 16#AB65;
   // GBK_TO_UNICODE[14165] := 16#73A1;
   // GBK_TO_UNICODE[14166] := 16#AB66;
   // GBK_TO_UNICODE[14167] := 16#73A3;
   // GBK_TO_UNICODE[14168] := 16#AB67;
   // GBK_TO_UNICODE[14169] := 16#73A4;
   // GBK_TO_UNICODE[14170] := 16#AB68;
   // GBK_TO_UNICODE[14171] := 16#73A5;
   // GBK_TO_UNICODE[14172] := 16#AB69;
   // GBK_TO_UNICODE[14173] := 16#73A6;
   // GBK_TO_UNICODE[14174] := 16#AB6A;
   // GBK_TO_UNICODE[14175] := 16#73A7;
   // GBK_TO_UNICODE[14176] := 16#AB6B;
   // GBK_TO_UNICODE[14177] := 16#73A8;
   // GBK_TO_UNICODE[14178] := 16#AB6C;
   // GBK_TO_UNICODE[14179] := 16#73AA;
   // GBK_TO_UNICODE[14180] := 16#AB6D;
   // GBK_TO_UNICODE[14181] := 16#73AC;
   // GBK_TO_UNICODE[14182] := 16#AB6E;
   // GBK_TO_UNICODE[14183] := 16#73AD;
   // GBK_TO_UNICODE[14184] := 16#AB6F;
   // GBK_TO_UNICODE[14185] := 16#73B1;
   // GBK_TO_UNICODE[14186] := 16#AB70;
   // GBK_TO_UNICODE[14187] := 16#73B4;
   // GBK_TO_UNICODE[14188] := 16#AB71;
   // GBK_TO_UNICODE[14189] := 16#73B5;
   // GBK_TO_UNICODE[14190] := 16#AB72;
   // GBK_TO_UNICODE[14191] := 16#73B6;
   // GBK_TO_UNICODE[14192] := 16#AB73;
   // GBK_TO_UNICODE[14193] := 16#73B8;
   // GBK_TO_UNICODE[14194] := 16#AB74;
   // GBK_TO_UNICODE[14195] := 16#73B9;
   // GBK_TO_UNICODE[14196] := 16#AB75;
   // GBK_TO_UNICODE[14197] := 16#73BC;
   // GBK_TO_UNICODE[14198] := 16#AB76;
   // GBK_TO_UNICODE[14199] := 16#73BD;
   // GBK_TO_UNICODE[14200] := 16#AB77;
   // GBK_TO_UNICODE[14201] := 16#73BE;
   // GBK_TO_UNICODE[14202] := 16#AB78;
   // GBK_TO_UNICODE[14203] := 16#73BF;
   // GBK_TO_UNICODE[14204] := 16#AB79;
   // GBK_TO_UNICODE[14205] := 16#73C1;
   // GBK_TO_UNICODE[14206] := 16#AB7A;
   // GBK_TO_UNICODE[14207] := 16#73C3;
   // GBK_TO_UNICODE[14208] := 16#AB7B;
   // GBK_TO_UNICODE[14209] := 16#73C4;
   // GBK_TO_UNICODE[14210] := 16#AB7C;
   // GBK_TO_UNICODE[14211] := 16#73C5;
   // GBK_TO_UNICODE[14212] := 16#AB7D;
   // GBK_TO_UNICODE[14213] := 16#73C6;
   // GBK_TO_UNICODE[14214] := 16#AB7E;
   // GBK_TO_UNICODE[14215] := 16#73C7;
   // GBK_TO_UNICODE[14216] := 16#AB80;
   // GBK_TO_UNICODE[14217] := 16#73CB;
   // GBK_TO_UNICODE[14218] := 16#AB81;
   // GBK_TO_UNICODE[14219] := 16#73CC;
   // GBK_TO_UNICODE[14220] := 16#AB82;
   // GBK_TO_UNICODE[14221] := 16#73CE;
   // GBK_TO_UNICODE[14222] := 16#AB83;
   // GBK_TO_UNICODE[14223] := 16#73D2;
   // GBK_TO_UNICODE[14224] := 16#AB84;
   // GBK_TO_UNICODE[14225] := 16#73D3;
   // GBK_TO_UNICODE[14226] := 16#AB85;
   // GBK_TO_UNICODE[14227] := 16#73D4;
   // GBK_TO_UNICODE[14228] := 16#AB86;
   // GBK_TO_UNICODE[14229] := 16#73D5;
   // GBK_TO_UNICODE[14230] := 16#AB87;
   // GBK_TO_UNICODE[14231] := 16#73D6;
   // GBK_TO_UNICODE[14232] := 16#AB88;
   // GBK_TO_UNICODE[14233] := 16#73D7;
   // GBK_TO_UNICODE[14234] := 16#AB89;
   // GBK_TO_UNICODE[14235] := 16#73D8;
   // GBK_TO_UNICODE[14236] := 16#AB8A;
   // GBK_TO_UNICODE[14237] := 16#73DA;
   // GBK_TO_UNICODE[14238] := 16#AB8B;
   // GBK_TO_UNICODE[14239] := 16#73DB;
   // GBK_TO_UNICODE[14240] := 16#AB8C;
   // GBK_TO_UNICODE[14241] := 16#73DC;
   // GBK_TO_UNICODE[14242] := 16#AB8D;
   // GBK_TO_UNICODE[14243] := 16#73DD;
   // GBK_TO_UNICODE[14244] := 16#AB8E;
   // GBK_TO_UNICODE[14245] := 16#73DF;
   // GBK_TO_UNICODE[14246] := 16#AB8F;
   // GBK_TO_UNICODE[14247] := 16#73E1;
   // GBK_TO_UNICODE[14248] := 16#AB90;
   // GBK_TO_UNICODE[14249] := 16#73E2;
   // GBK_TO_UNICODE[14250] := 16#AB91;
   // GBK_TO_UNICODE[14251] := 16#73E3;
   // GBK_TO_UNICODE[14252] := 16#AB92;
   // GBK_TO_UNICODE[14253] := 16#73E4;
   // GBK_TO_UNICODE[14254] := 16#AB93;
   // GBK_TO_UNICODE[14255] := 16#73E6;
   // GBK_TO_UNICODE[14256] := 16#AB94;
   // GBK_TO_UNICODE[14257] := 16#73E8;
   // GBK_TO_UNICODE[14258] := 16#AB95;
   // GBK_TO_UNICODE[14259] := 16#73EA;
   // GBK_TO_UNICODE[14260] := 16#AB96;
   // GBK_TO_UNICODE[14261] := 16#73EB;
   // GBK_TO_UNICODE[14262] := 16#AB97;
   // GBK_TO_UNICODE[14263] := 16#73EC;
   // GBK_TO_UNICODE[14264] := 16#AB98;
   // GBK_TO_UNICODE[14265] := 16#73EE;
   // GBK_TO_UNICODE[14266] := 16#AB99;
   // GBK_TO_UNICODE[14267] := 16#73EF;
   // GBK_TO_UNICODE[14268] := 16#AB9A;
   // GBK_TO_UNICODE[14269] := 16#73F0;
   // GBK_TO_UNICODE[14270] := 16#AB9B;
   // GBK_TO_UNICODE[14271] := 16#73F1;
   // GBK_TO_UNICODE[14272] := 16#AB9C;
   // GBK_TO_UNICODE[14273] := 16#73F3;
   // GBK_TO_UNICODE[14274] := 16#AB9D;
   // GBK_TO_UNICODE[14275] := 16#73F4;
   // GBK_TO_UNICODE[14276] := 16#AB9E;
   // GBK_TO_UNICODE[14277] := 16#73F5;
   // GBK_TO_UNICODE[14278] := 16#AB9F;
   // GBK_TO_UNICODE[14279] := 16#73F6;
   // GBK_TO_UNICODE[14280] := 16#ABA0;
   // GBK_TO_UNICODE[14281] := 16#73F7;
   // GBK_TO_UNICODE[14282] := 16#AC40;
   // GBK_TO_UNICODE[14283] := 16#73F8;
   // GBK_TO_UNICODE[14284] := 16#AC41;
   // GBK_TO_UNICODE[14285] := 16#73F9;
   // GBK_TO_UNICODE[14286] := 16#AC42;
   // GBK_TO_UNICODE[14287] := 16#73FA;
   // GBK_TO_UNICODE[14288] := 16#AC43;
   // GBK_TO_UNICODE[14289] := 16#73FB;
   // GBK_TO_UNICODE[14290] := 16#AC44;
   // GBK_TO_UNICODE[14291] := 16#73FC;
   // GBK_TO_UNICODE[14292] := 16#AC45;
   // GBK_TO_UNICODE[14293] := 16#73FD;
   // GBK_TO_UNICODE[14294] := 16#AC46;
   // GBK_TO_UNICODE[14295] := 16#73FE;
   // GBK_TO_UNICODE[14296] := 16#AC47;
   // GBK_TO_UNICODE[14297] := 16#73FF;
   // GBK_TO_UNICODE[14298] := 16#AC48;
   // GBK_TO_UNICODE[14299] := 16#7400;
   // GBK_TO_UNICODE[14300] := 16#AC49;
   // GBK_TO_UNICODE[14301] := 16#7401;
   // GBK_TO_UNICODE[14302] := 16#AC4A;
   // GBK_TO_UNICODE[14303] := 16#7402;
   // GBK_TO_UNICODE[14304] := 16#AC4B;
   // GBK_TO_UNICODE[14305] := 16#7404;
   // GBK_TO_UNICODE[14306] := 16#AC4C;
   // GBK_TO_UNICODE[14307] := 16#7407;
   // GBK_TO_UNICODE[14308] := 16#AC4D;
   // GBK_TO_UNICODE[14309] := 16#7408;
   // GBK_TO_UNICODE[14310] := 16#AC4E;
   // GBK_TO_UNICODE[14311] := 16#740B;
   // GBK_TO_UNICODE[14312] := 16#AC4F;
   // GBK_TO_UNICODE[14313] := 16#740C;
   // GBK_TO_UNICODE[14314] := 16#AC50;
   // GBK_TO_UNICODE[14315] := 16#740D;
   // GBK_TO_UNICODE[14316] := 16#AC51;
   // GBK_TO_UNICODE[14317] := 16#740E;
   // GBK_TO_UNICODE[14318] := 16#AC52;
   // GBK_TO_UNICODE[14319] := 16#7411;
   // GBK_TO_UNICODE[14320] := 16#AC53;
   // GBK_TO_UNICODE[14321] := 16#7412;
   // GBK_TO_UNICODE[14322] := 16#AC54;
   // GBK_TO_UNICODE[14323] := 16#7413;
   // GBK_TO_UNICODE[14324] := 16#AC55;
   // GBK_TO_UNICODE[14325] := 16#7414;
   // GBK_TO_UNICODE[14326] := 16#AC56;
   // GBK_TO_UNICODE[14327] := 16#7415;
   // GBK_TO_UNICODE[14328] := 16#AC57;
   // GBK_TO_UNICODE[14329] := 16#7416;
   // GBK_TO_UNICODE[14330] := 16#AC58;
   // GBK_TO_UNICODE[14331] := 16#7417;
   // GBK_TO_UNICODE[14332] := 16#AC59;
   // GBK_TO_UNICODE[14333] := 16#7418;
   // GBK_TO_UNICODE[14334] := 16#AC5A;
   // GBK_TO_UNICODE[14335] := 16#7419;
   // GBK_TO_UNICODE[14336] := 16#AC5B;
   // GBK_TO_UNICODE[14337] := 16#741C;
   // GBK_TO_UNICODE[14338] := 16#AC5C;
   // GBK_TO_UNICODE[14339] := 16#741D;
   // GBK_TO_UNICODE[14340] := 16#AC5D;
   // GBK_TO_UNICODE[14341] := 16#741E;
   // GBK_TO_UNICODE[14342] := 16#AC5E;
   // GBK_TO_UNICODE[14343] := 16#741F;
   // GBK_TO_UNICODE[14344] := 16#AC5F;
   // GBK_TO_UNICODE[14345] := 16#7420;
   // GBK_TO_UNICODE[14346] := 16#AC60;
   // GBK_TO_UNICODE[14347] := 16#7421;
   // GBK_TO_UNICODE[14348] := 16#AC61;
   // GBK_TO_UNICODE[14349] := 16#7423;
   // GBK_TO_UNICODE[14350] := 16#AC62;
   // GBK_TO_UNICODE[14351] := 16#7424;
   // GBK_TO_UNICODE[14352] := 16#AC63;
   // GBK_TO_UNICODE[14353] := 16#7427;
   // GBK_TO_UNICODE[14354] := 16#AC64;
   // GBK_TO_UNICODE[14355] := 16#7429;
   // GBK_TO_UNICODE[14356] := 16#AC65;
   // GBK_TO_UNICODE[14357] := 16#742B;
   // GBK_TO_UNICODE[14358] := 16#AC66;
   // GBK_TO_UNICODE[14359] := 16#742D;
   // GBK_TO_UNICODE[14360] := 16#AC67;
   // GBK_TO_UNICODE[14361] := 16#742F;
   // GBK_TO_UNICODE[14362] := 16#AC68;
   // GBK_TO_UNICODE[14363] := 16#7431;
   // GBK_TO_UNICODE[14364] := 16#AC69;
   // GBK_TO_UNICODE[14365] := 16#7432;
   // GBK_TO_UNICODE[14366] := 16#AC6A;
   // GBK_TO_UNICODE[14367] := 16#7437;
   // GBK_TO_UNICODE[14368] := 16#AC6B;
   // GBK_TO_UNICODE[14369] := 16#7438;
   // GBK_TO_UNICODE[14370] := 16#AC6C;
   // GBK_TO_UNICODE[14371] := 16#7439;
   // GBK_TO_UNICODE[14372] := 16#AC6D;
   // GBK_TO_UNICODE[14373] := 16#743A;
   // GBK_TO_UNICODE[14374] := 16#AC6E;
   // GBK_TO_UNICODE[14375] := 16#743B;
   // GBK_TO_UNICODE[14376] := 16#AC6F;
   // GBK_TO_UNICODE[14377] := 16#743D;
   // GBK_TO_UNICODE[14378] := 16#AC70;
   // GBK_TO_UNICODE[14379] := 16#743E;
   // GBK_TO_UNICODE[14380] := 16#AC71;
   // GBK_TO_UNICODE[14381] := 16#743F;
   // GBK_TO_UNICODE[14382] := 16#AC72;
   // GBK_TO_UNICODE[14383] := 16#7440;
   // GBK_TO_UNICODE[14384] := 16#AC73;
   // GBK_TO_UNICODE[14385] := 16#7442;
   // GBK_TO_UNICODE[14386] := 16#AC74;
   // GBK_TO_UNICODE[14387] := 16#7443;
   // GBK_TO_UNICODE[14388] := 16#AC75;
   // GBK_TO_UNICODE[14389] := 16#7444;
   // GBK_TO_UNICODE[14390] := 16#AC76;
   // GBK_TO_UNICODE[14391] := 16#7445;
   // GBK_TO_UNICODE[14392] := 16#AC77;
   // GBK_TO_UNICODE[14393] := 16#7446;
   // GBK_TO_UNICODE[14394] := 16#AC78;
   // GBK_TO_UNICODE[14395] := 16#7447;
   // GBK_TO_UNICODE[14396] := 16#AC79;
   // GBK_TO_UNICODE[14397] := 16#7448;
   // GBK_TO_UNICODE[14398] := 16#AC7A;
   // GBK_TO_UNICODE[14399] := 16#7449;
   // GBK_TO_UNICODE[14400] := 16#AC7B;
   // GBK_TO_UNICODE[14401] := 16#744A;
   // GBK_TO_UNICODE[14402] := 16#AC7C;
   // GBK_TO_UNICODE[14403] := 16#744B;
   // GBK_TO_UNICODE[14404] := 16#AC7D;
   // GBK_TO_UNICODE[14405] := 16#744C;
   // GBK_TO_UNICODE[14406] := 16#AC7E;
   // GBK_TO_UNICODE[14407] := 16#744D;
   // GBK_TO_UNICODE[14408] := 16#AC80;
   // GBK_TO_UNICODE[14409] := 16#744E;
   // GBK_TO_UNICODE[14410] := 16#AC81;
   // GBK_TO_UNICODE[14411] := 16#744F;
   // GBK_TO_UNICODE[14412] := 16#AC82;
   // GBK_TO_UNICODE[14413] := 16#7450;
   // GBK_TO_UNICODE[14414] := 16#AC83;
   // GBK_TO_UNICODE[14415] := 16#7451;
   // GBK_TO_UNICODE[14416] := 16#AC84;
   // GBK_TO_UNICODE[14417] := 16#7452;
   // GBK_TO_UNICODE[14418] := 16#AC85;
   // GBK_TO_UNICODE[14419] := 16#7453;
   // GBK_TO_UNICODE[14420] := 16#AC86;
   // GBK_TO_UNICODE[14421] := 16#7454;
   // GBK_TO_UNICODE[14422] := 16#AC87;
   // GBK_TO_UNICODE[14423] := 16#7456;
   // GBK_TO_UNICODE[14424] := 16#AC88;
   // GBK_TO_UNICODE[14425] := 16#7458;
   // GBK_TO_UNICODE[14426] := 16#AC89;
   // GBK_TO_UNICODE[14427] := 16#745D;
   // GBK_TO_UNICODE[14428] := 16#AC8A;
   // GBK_TO_UNICODE[14429] := 16#7460;
   // GBK_TO_UNICODE[14430] := 16#AC8B;
   // GBK_TO_UNICODE[14431] := 16#7461;
   // GBK_TO_UNICODE[14432] := 16#AC8C;
   // GBK_TO_UNICODE[14433] := 16#7462;
   // GBK_TO_UNICODE[14434] := 16#AC8D;
   // GBK_TO_UNICODE[14435] := 16#7463;
   // GBK_TO_UNICODE[14436] := 16#AC8E;
   // GBK_TO_UNICODE[14437] := 16#7464;
   // GBK_TO_UNICODE[14438] := 16#AC8F;
   // GBK_TO_UNICODE[14439] := 16#7465;
   // GBK_TO_UNICODE[14440] := 16#AC90;
   // GBK_TO_UNICODE[14441] := 16#7466;
   // GBK_TO_UNICODE[14442] := 16#AC91;
   // GBK_TO_UNICODE[14443] := 16#7467;
   // GBK_TO_UNICODE[14444] := 16#AC92;
   // GBK_TO_UNICODE[14445] := 16#7468;
   // GBK_TO_UNICODE[14446] := 16#AC93;
   // GBK_TO_UNICODE[14447] := 16#7469;
   // GBK_TO_UNICODE[14448] := 16#AC94;
   // GBK_TO_UNICODE[14449] := 16#746A;
   // GBK_TO_UNICODE[14450] := 16#AC95;
   // GBK_TO_UNICODE[14451] := 16#746B;
   // GBK_TO_UNICODE[14452] := 16#AC96;
   // GBK_TO_UNICODE[14453] := 16#746C;
   // GBK_TO_UNICODE[14454] := 16#AC97;
   // GBK_TO_UNICODE[14455] := 16#746E;
   // GBK_TO_UNICODE[14456] := 16#AC98;
   // GBK_TO_UNICODE[14457] := 16#746F;
   // GBK_TO_UNICODE[14458] := 16#AC99;
   // GBK_TO_UNICODE[14459] := 16#7471;
   // GBK_TO_UNICODE[14460] := 16#AC9A;
   // GBK_TO_UNICODE[14461] := 16#7472;
   // GBK_TO_UNICODE[14462] := 16#AC9B;
   // GBK_TO_UNICODE[14463] := 16#7473;
   // GBK_TO_UNICODE[14464] := 16#AC9C;
   // GBK_TO_UNICODE[14465] := 16#7474;
   // GBK_TO_UNICODE[14466] := 16#AC9D;
   // GBK_TO_UNICODE[14467] := 16#7475;
   // GBK_TO_UNICODE[14468] := 16#AC9E;
   // GBK_TO_UNICODE[14469] := 16#7478;
   // GBK_TO_UNICODE[14470] := 16#AC9F;
   // GBK_TO_UNICODE[14471] := 16#7479;
   // GBK_TO_UNICODE[14472] := 16#ACA0;
   // GBK_TO_UNICODE[14473] := 16#747A;
   // GBK_TO_UNICODE[14474] := 16#AD40;
   // GBK_TO_UNICODE[14475] := 16#747B;
   // GBK_TO_UNICODE[14476] := 16#AD41;
   // GBK_TO_UNICODE[14477] := 16#747C;
   // GBK_TO_UNICODE[14478] := 16#AD42;
   // GBK_TO_UNICODE[14479] := 16#747D;
   // GBK_TO_UNICODE[14480] := 16#AD43;
   // GBK_TO_UNICODE[14481] := 16#747F;
   // GBK_TO_UNICODE[14482] := 16#AD44;
   // GBK_TO_UNICODE[14483] := 16#7482;
   // GBK_TO_UNICODE[14484] := 16#AD45;
   // GBK_TO_UNICODE[14485] := 16#7484;
   // GBK_TO_UNICODE[14486] := 16#AD46;
   // GBK_TO_UNICODE[14487] := 16#7485;
   // GBK_TO_UNICODE[14488] := 16#AD47;
   // GBK_TO_UNICODE[14489] := 16#7486;
   // GBK_TO_UNICODE[14490] := 16#AD48;
   // GBK_TO_UNICODE[14491] := 16#7488;
   // GBK_TO_UNICODE[14492] := 16#AD49;
   // GBK_TO_UNICODE[14493] := 16#7489;
   // GBK_TO_UNICODE[14494] := 16#AD4A;
   // GBK_TO_UNICODE[14495] := 16#748A;
   // GBK_TO_UNICODE[14496] := 16#AD4B;
   // GBK_TO_UNICODE[14497] := 16#748C;
   // GBK_TO_UNICODE[14498] := 16#AD4C;
   // GBK_TO_UNICODE[14499] := 16#748D;
   // GBK_TO_UNICODE[14500] := 16#AD4D;
   // GBK_TO_UNICODE[14501] := 16#748F;
   // GBK_TO_UNICODE[14502] := 16#AD4E;
   // GBK_TO_UNICODE[14503] := 16#7491;
   // GBK_TO_UNICODE[14504] := 16#AD4F;
   // GBK_TO_UNICODE[14505] := 16#7492;
   // GBK_TO_UNICODE[14506] := 16#AD50;
   // GBK_TO_UNICODE[14507] := 16#7493;
   // GBK_TO_UNICODE[14508] := 16#AD51;
   // GBK_TO_UNICODE[14509] := 16#7494;
   // GBK_TO_UNICODE[14510] := 16#AD52;
   // GBK_TO_UNICODE[14511] := 16#7495;
   // GBK_TO_UNICODE[14512] := 16#AD53;
   // GBK_TO_UNICODE[14513] := 16#7496;
   // GBK_TO_UNICODE[14514] := 16#AD54;
   // GBK_TO_UNICODE[14515] := 16#7497;
   // GBK_TO_UNICODE[14516] := 16#AD55;
   // GBK_TO_UNICODE[14517] := 16#7498;
   // GBK_TO_UNICODE[14518] := 16#AD56;
   // GBK_TO_UNICODE[14519] := 16#7499;
   // GBK_TO_UNICODE[14520] := 16#AD57;
   // GBK_TO_UNICODE[14521] := 16#749A;
   // GBK_TO_UNICODE[14522] := 16#AD58;
   // GBK_TO_UNICODE[14523] := 16#749B;
   // GBK_TO_UNICODE[14524] := 16#AD59;
   // GBK_TO_UNICODE[14525] := 16#749D;
   // GBK_TO_UNICODE[14526] := 16#AD5A;
   // GBK_TO_UNICODE[14527] := 16#749F;
   // GBK_TO_UNICODE[14528] := 16#AD5B;
   // GBK_TO_UNICODE[14529] := 16#74A0;
   // GBK_TO_UNICODE[14530] := 16#AD5C;
   // GBK_TO_UNICODE[14531] := 16#74A1;
   // GBK_TO_UNICODE[14532] := 16#AD5D;
   // GBK_TO_UNICODE[14533] := 16#74A2;
   // GBK_TO_UNICODE[14534] := 16#AD5E;
   // GBK_TO_UNICODE[14535] := 16#74A3;
   // GBK_TO_UNICODE[14536] := 16#AD5F;
   // GBK_TO_UNICODE[14537] := 16#74A4;
   // GBK_TO_UNICODE[14538] := 16#AD60;
   // GBK_TO_UNICODE[14539] := 16#74A5;
   // GBK_TO_UNICODE[14540] := 16#AD61;
   // GBK_TO_UNICODE[14541] := 16#74A6;
   // GBK_TO_UNICODE[14542] := 16#AD62;
   // GBK_TO_UNICODE[14543] := 16#74AA;
   // GBK_TO_UNICODE[14544] := 16#AD63;
   // GBK_TO_UNICODE[14545] := 16#74AB;
   // GBK_TO_UNICODE[14546] := 16#AD64;
   // GBK_TO_UNICODE[14547] := 16#74AC;
   // GBK_TO_UNICODE[14548] := 16#AD65;
   // GBK_TO_UNICODE[14549] := 16#74AD;
   // GBK_TO_UNICODE[14550] := 16#AD66;
   // GBK_TO_UNICODE[14551] := 16#74AE;
   // GBK_TO_UNICODE[14552] := 16#AD67;
   // GBK_TO_UNICODE[14553] := 16#74AF;
   // GBK_TO_UNICODE[14554] := 16#AD68;
   // GBK_TO_UNICODE[14555] := 16#74B0;
   // GBK_TO_UNICODE[14556] := 16#AD69;
   // GBK_TO_UNICODE[14557] := 16#74B1;
   // GBK_TO_UNICODE[14558] := 16#AD6A;
   // GBK_TO_UNICODE[14559] := 16#74B2;
   // GBK_TO_UNICODE[14560] := 16#AD6B;
   // GBK_TO_UNICODE[14561] := 16#74B3;
   // GBK_TO_UNICODE[14562] := 16#AD6C;
   // GBK_TO_UNICODE[14563] := 16#74B4;
   // GBK_TO_UNICODE[14564] := 16#AD6D;
   // GBK_TO_UNICODE[14565] := 16#74B5;
   // GBK_TO_UNICODE[14566] := 16#AD6E;
   // GBK_TO_UNICODE[14567] := 16#74B6;
